# B&R Automation Studio project BR_ZBM1 (part 3)

#### SC_9Init.st - Initialization code
```iecst
(********************************************************************
 * COPYRIGHT --
 ********************************************************************
 * Program: SC_2
 * File: SC_2Init.st
 * Author: ronspa
 * Created: February 16, 2015
 ********************************************************************
 * Implementation of program SC_2
 ********************************************************************)

PROGRAM _INIT

	i := 8;

END_PROGRAM
```

- SC.st (reference to Logical/BunchUnits/SC_Ref/SC.st)

- SC.var (reference to Logical/BunchUnits/SC_Ref/SC.var)

### Program Logical/BunchUnits/BU_10 (IEC) - Program for Bunch Unit 10

#### BU_10Init.st - Initialization code
```iecst
(********************************************************************
 * COPYRIGHT --
 ********************************************************************
 * Program: BU_1
 * File: BU_1Init.st
 * Author: ronspa
 * Created: Januari 12, 2015
 ********************************************************************
 * Implementation of program BU_1
 ********************************************************************)

PROGRAM _INIT

	i := 9;

	BU[i].typInterface.Status := BU_ST_DISABLED;
	BU[i].usChainPos := SHFTREG.uiBunchUnitPosition[i] - 1; // Because position is 0!!!

	// For TESTING RSP 23-12-2014

	//Enable 'FI'
	BU[i].typBunchBelts.command.bEnabledStop := TRUE;
	//Bepaal draairichting
	BU[i].typBunchBelts.command.bRunReverse := FALSE;
	BU[i].typSettings.usTimingBU16 := 14; // Pos=0 ->

END_PROGRAM
```

- BunchUnit.st (reference to Logical/BunchUnits/BU_Ref/BunchUnit.st)

- BunchUnit.var (reference to Logical/BunchUnits/BU_Ref/BunchUnit.var)

### Program Logical/BunchUnits/SC_10 (IEC) - Program for Servo 10

#### SC_10Init.st - Initialization code
```iecst
(********************************************************************
 * COPYRIGHT --
 ********************************************************************
 * Program: SC_2
 * File: SC_2Init.st
 * Author: ronspa
 * Created: February 16, 2015
 ********************************************************************
 * Implementation of program SC_2
 ********************************************************************)

PROGRAM _INIT

	i := 9;

END_PROGRAM
```

- SC.st (reference to Logical/BunchUnits/SC_Ref/SC.st)

- SC.var (reference to Logical/BunchUnits/SC_Ref/SC.var)

### Package Logical/Exceptionhandling - All error codes and exceptions

### Program Logical/Exceptionhandling/ErrorHandling (IEC) - Program

#### ErrorHandling.st - Implementation code
```iecst
(********************************************************************
 * COPYRIGHT --
 ********************************************************************
 * Program: ErrorHandling
 * File: ErrorHandling.st
 * Author: jorkes
 * Created: July 21, 2014
 ********************************************************************
 * Implementation of program ErrorHandling
 ********************************************************************)

PROGRAM _INIT

(* TODO : Add your code here *)

END_PROGRAM

PROGRAM _CYCLIC
	tonHeartBeat( IN:= NOT(EDGE(bHeartBeat)), PT:= INT_TO_TIME(Settings.HeartBeatTime));
	IF EDGE(tonHeartBeat.Q ) THEN
		// LOG
		IF(tonHeartBeat.Q) THEN
			AsArLogWrite_Failed(enable := TRUE, ident := arlogBASE_USER_LOG_IDENT, logLevel := 1, errornr := 50001, mem := 0, len := 0, asciiString :=  ADR('Heart beat failed!!!!'));
		ELSE
			AsArLogWrite_Restored(enable := TRUE, ident := arlogBASE_USER_LOG_IDENT, logLevel := 1, errornr := 50001, mem := 0, len := 0, asciiString :=  ADR('Heart beat active again'));
		END_IF
	END_IF

	IF MCU.typIN.bEmergencyStop THEN
		ErrorState := EMERGENCYSTOP;
	ELSIF MCU.typIN.bDoorOpen THEN
		ErrorState := DOOROPEN;
	ELSIF MCU.typIN.bServiceMode THEN
		ErrorState := SERVICEMODE;
	ELSIF MCU.typIN.bAirpressure THEN
		ErrorState := AIRPRESSURE;
	ELSIF MCU.typIN.bBinder THEN
		ErrorState := BINDER;
	ELSE
		ErrorState := OK;
	END_IF

	//enumError
	CASE ErrorState OF
		0: bGblRun := FALSE;//EmergencyStop
		1: //AirPressure
		2: //DoorOpen
		3: //MotorMalfunction
		4: //Communication
		5: //Binder
		6: //ServiceMode
	END_CASE

END_PROGRAM
```

#### ErrorHandling.var - Local variables
```iecst
(********************************************************************
 * COPYRIGHT --
 ********************************************************************
 * Program: ErrorHandling
 * File: ErrorHandling.var
 * Author: jorkes
 * Created: July 21, 2014
 ********************************************************************
 * Local variables of program ErrorHandling
 ********************************************************************)
VAR
	tonHeartBeat : TON;
	bHeartBeat : BOOL;
	AsArLogWrite_Failed : AsArLogWrite := (0);
	AsArLogWrite_Restored : AsArLogWrite := (0);
	LogMsg : STRING[80];
END_VAR
```

### Program Logical/Exceptionhandling/can_diag (IEC) - Program

#### can_diag.st - Implementation code
```iecst
(********************************************************************
 * COPYRIGHT -- Bernecker + Rainer
 ********************************************************************
 * Program: can_diag
 * File: can_diag.st
 * Author: fleischerm
 * Created: February 02, 2015
 ********************************************************************
 * Implementation of program can_diag
 ********************************************************************)

//******************************************************************
//
//	i n i t
//
//******************************************************************
PROGRAM _INIT

//******************************************************************
// RCX Common Status & Errors Codes
//------------------------------------------------------------------
// variable for the following error codes is -> x20if1041map.comError
//------------------------------------------------------------------
//	RCX_S_OK						0x00000000	Success, Status Okay
//	RCX_E_FAIL						0xC0000001 	Fail
//	RCX_E_UNEXPECTED				0xC0000002	Unexpected
//	RCX_E_OUTOFMEMORY				0xC0000003 	Out OF Memory
//	RCX_E_UNKNOWN_COMMAND			0xC0000004	Unknown Command
//	RCX_E_UNKNOWN_DESTINATION		0xC0000005	Unknown Destination
//	RCX_E_UNKNOWN_DESTINATION_ID	0xC0000006	Unknown Destination ID
//	RCX_E_INVALID_PACKET_LEN		0xC0000007	Invalid Packet Length
//	RCX_E_INVALID_EXTENSION			0xC0000008	Invalid Extension
//	RCX_E_INVALID_PARAMETER			0xC0000009	Invalid Parameter
//	RCX_E_WATCHDOG_TIMEOUT			0xC000000C	Watchdog Timeout
//	RCX_E_INVALID_LIST_TYPE			0xC000000D	Invalid List Type
//	RCX_E_UNKNOWN_HANDLE			0xC000000E	Unknown Handle
//	RCX_E_PACKET_OUT_OF_SEQ			0xC000000F	Out OF Sequence
//	RCX_E_PACKET_OUT_OF_MEMORY		0xC0000010	Out OF Memory
//	RCX_E_QUE_PACKETDONE			0xC0000011	Queue Packet Done
//	RCX_E_QUE_SENDPACKET			0xC0000012	Queue Send Packet
//	RCX_E_POOL_PACKET_GET			0xC0000013	Pool Packet Get
//	RCX_E_POOL_GET_LOAD				0xC0000015	Pool Get Load
//	RCX_E_REQUEST_RUNNING			0xC000001A	Request Already Running
//	RCX_E_INIT_FAULT				0xC0000100	Initialization Fault
//	RCX_E_DATABASE_ACCESS_FAILED	0xC0000101	Database ACCESS Failed
//	RCX_E_NOT_CONFIGURED			0xC0000119	NOT Configured
//	RCX_E_CONFIGURATION_FAULT		0xC0000120	Configuration Fault
//	RCX_E_INCONSISTENT_DATA_SET		0xC0000121	Inconsistent Data Set
//	RCX_E_DATA_SET_MISMATCH			0xC0000122	Data Set Mismatch
//	RCX_E_INSUFFICIENT_LICENSE		0xC0000123	Insufficient License
//	RCX_E_PARAMETER_ERROR			0xC0000124	Parameter Error
//	RCX_E_INVALID_NETWORK_ADDRESS	0xC0000125	Invalid Network Address
//	RCX_E_NO_SECURITY_MEMORY		0xC0000126	No Security Memory
//	RCX_E_NETWORK_FAULT				0xC0000140	Network Fault
//	RCX_E_CONNECTION_CLOSED			0xC0000141	Connection Closed
//	RCX_E_CONNECTION_TIMEOUT		0xC0000142	Connection Timeout
//	RCX_E_LONELY_NETWORK			0xC0000143	Lonely Network
//	RCX_E_DUPLICATE_NODE			0xC0000144	Duplicate Node
//	RCX_E_CABLE_DISCONNECT			0xC0000145	Cable Disconnected
//	RCX_E_BUS_OFF					0xC0000180	Network Node Bus Off
//	RCX_E_CONFIG_LOCKED				0xC0000181	Configuration Locked
//	RCX_E_APPLICATION_NOT_READY		0xC0000182	Application NOT Ready
//	RCX_E_TIMER_APPL_PACKET_SENT	0xC002000C	Timer App Packet Sent
//******************************************************************

//******************************************************************
// RCX Status & Error Codes Slave State
//------------------------------------------------------------------
// variable for the following error codes is -> x20if1041map.slaveState
//------------------------------------------------------------------
//	RCX_SLAVE_STATE_UNDEFINED		0x00000000	UNDEFINED
//	RCX_SLAVE_STATE_OK				0x00000001	OK
//	RCX_SLAVE_STATE_FAILED			0x00000002	FAILED (at least one slave)
//******************************************************************

//******************************************************************
// init some variables
//******************************************************************
step									:= 255;
getDiagInfo								:= FALSE;

END_PROGRAM

//******************************************************************
//
//	c y c l i c
//
//******************************************************************
PROGRAM _CYCLIC

	//******************************************************************************
	// Havatec global used data structure for OPC, VIS and Control
	//**************************************************************
	BU[0];

	//******************************************************************************
	// CANopen Master -> X20IF1041-1
	// get data structure from the I/O mapping
	//**************************************************************
	CASE x20if1041map.comState OF
	//**************************************************************
	0: 	// Unkown
	2:	// Stop
	3:	// Standby
	4:	// Operate
	END_CASE

	//**************************************************************
	CASE x20if1041map.comError OF
	//**************************************************************
	16#C0000140:	// General communication error (this error will occur if at least one slave in the CAN network isn't working)
	16#C0000142:	// Timeout while establishing connection
	16#C0000144:	// Repeated node number found in CAN network
	16#C0000145:	// CAN cable has been disconnected
	END_CASE

	//**************************************************************
	CASE x20if1041map.slaveState OF
	//**************************************************************
	0: 	// Undefined
	1:	// OK
	2:	// Failed
	3:	// Warning
	END_CASE

	//******************************************************************************
	// Servo Unit I/O mapping
	// - Module OK signal
	// - will be FALSE on network or cable error
	//**************************************************************
	IF (BU[0].typServo.bOnLine = FALSE) THEN							// a better check is to wait a certain time before the error is TRUE
		;
	END_IF

	//**************************************************************
	// Servo Unit I/O mapping
	// - Festo drive in error state
 	// -- 16#08 means drive is faulty
	//**************************************************************
	IF (BU[0].typServo.packed.SCON.3 = TRUE) THEN
		getDiagInfo						:= TRUE;
	ELSE
		getDiagInfo						:= FALSE;
	END_IF

	//**************************************************************
	IF EDGEPOS(getDiagInfo) THEN
		step							:= 2;							// next step -
	END_IF

	//******************************************************************************
	// call different function blocks
	//**************************************************************
	CASE step OF														// case function switch of
	//**************************************************************
	1:	// get emergency telegrams
		//**********************************************************
		nxcomRecvEmcyDev_0.enable 		:= TRUE;						// enable function block
		nxcomRecvEmcyDev_0.pDevice 		:= ADR('SS1.IF1');				// CANopen interface address
		nxcomRecvEmcyDev_0.node 		:= 3;							// node number (client address)
		nxcomRecvEmcyDev_0.flags		:= nxcomFLAG_PEEK;				// means: Don't remove node from the diagnostics list
		nxcomRecvEmcyDev_0.pEmcyData	:= ADR(emcyTelegram);			// pointer to an array of 5 emergency telegrams with 8 bytes each
		nxcomRecvEmcyDev_0();											// call function block instance

		//**********************************************************
		CASE nxcomRecvEmcyDev_0.status OF								// case function switch of
		//**********************************************************
		65535:	// ERR_BUSY
			//******************************************************
			;															// wait for different status
		//**********************************************************
		0:		// ERR_OK
			//******************************************************
			nxcomRecvEmcyDev_0.coStatus;								// see help file for the nxcomGetDiag function block
			nxcomRecvEmcyDev_0.emcyCount;								// ...
			//******************************************************
			step						:= 255;							// next step -
		ELSE
			//******************************************************
			step						:= 255;							// next step -
		END_CASE

	//**************************************************************
	2:	// read the diagnostics for the specified node
		// ->
		// -> inclusive the last b5 emergency telegrams
		// ->
		//**********************************************************
		nxcomGetDiag_0.enable 			:= TRUE;						// enable function block
		nxcomGetDiag_0.pDevice 			:= ADR('SS1.IF1');				// CANopen interface address
		nxcomGetDiag_0.node 			:= 3;							// node number (client address)
		nxcomGetDiag_0.flags 			:= nxcomFLAG_PEEK;				// means: Don't remove node from the diagnostics list
		nxcomGetDiag_0.pEmcyData 		:= ADR(emcyTelegram);			// pointer to an array of 5 emergency telegrams with 8 bytes each
		nxcomGetDiag_0();												// call function block instance

		//**********************************************************
		CASE nxcomGetDiag_0.status OF									// case function switch of
		//**********************************************************
		65535:	// ERR_BUSY
			//******************************************************
			;															// wait for different status
		//**********************************************************
		0:		// ERR_OK
			//******************************************************
			nxcomGetDiag_0.coStatus;									// see help file for the nxcomGetDiag function block
			nxcomGetDiag_0.nodeFlags;									// ...
			nxcomGetDiag_0.lastDiagInfo;								// ...
			nxcomGetDiag_0.devType;										// ...
			nxcomGetDiag_0.nmtState;									// ...
			nxcomGetDiag_0.emcyCount;									// Number of actually read emergency telegrams.
			//******************************************************
			step						:= 255;							// next step -
		ELSE
			//******************************************************
			step						:= 255;							// next step -
		END_CASE
	ELSE
		//**********************************************************
		step							:= 255;							// next step -
	END_CASE

END_PROGRAM

//******************************************************************
//
//	e x i t
//
//******************************************************************
PROGRAM _EXIT

//******************************************************************
// TODO : Add your code here
//******************************************************************
nxcomRecvEmcyDev_0.enable 				:= FALSE;						// disable function block on exit
nxcomRecvEmcyDev_0();													// call function block instance

//******************************************************************
nxcomGetDiag_0.enable 					:= FALSE;						// disable function block on exit
nxcomGetDiag_0();														// call function block instance

END_PROGRAM
```

#### can_diag.typ - Local data types
```iecst
(********************************************************************
 * COPYRIGHT -- Bernecker + Rainer
 ********************************************************************
 * Program: can_diag
 * File: can_diag.typ
 * Author: fleischerm
 * Created: February 02, 2015
 ********************************************************************
 * Local data types of program can_diag
 ********************************************************************)

TYPE
	local_if1041_map : 	STRUCT
		comCOS : UDINT;
		comState : UDINT;
		comError : UDINT;
		version : UINT;
		watchdogTimeout : UINT;
		watchdogHost : UDINT;
		errorCount : UDINT;
		errorLogIndicator : UDINT;
		slaveState : UDINT;
		slaveErrorLogIndicator : UDINT;
		slavesConfigured : UDINT;
		slavesActive : UDINT;
		slavesFaulted : UDINT;
	END_STRUCT;
END_TYPE
```

#### can_diag.var - Local variables
```iecst
(********************************************************************
 * COPYRIGHT -- Bernecker + Rainer
 ********************************************************************
 * Program: can_diag
 * File: can_diag.var
 * Author: fleischerm
 * Created: February 02, 2015
 ********************************************************************
 * Local variables of program can_diag
 ********************************************************************)
VAR
	getDiagInfo : BOOL;
	step : USINT;
	x20if1041map : local_if1041_map;
	emcyTelegram : nxcomEmcyTelegrams_t;
	nxcomGetDiag_0 : nxcomGetDiag;
	nxcomRecvEmcyDev_0 : nxcomRecvEmcyDev;
END_VAR
```

- Visualisation Logical/Visualisation (not shown)

### Package Logical/Docs - Package

### ToDo.txt
```
In BunchUnit Ref is de aanstuur tijde van de puls aangepast van 100 -> 1000 voor test.

Bij tijdelijke code van Ronald staat de aanduiding RSPA, dit moet voor de uit eindelijk versie recht gezet worden.

Lijst van openstaande punten:

- Het afvoer bit implementeren zodat de BU geleegd kan worden.
- De timing voor de BunchBelt control in valiabele zetten
- CAN-bus communicatie check
- Keep alive met OPC implementeren, ter indicatie of de PC leeft (Actie bedenken indien dood)
- Enable koppelen aan VNC GUI, zodat met minder BU's gewerkt kan worden.
- GUI aanpassen zodat deze door de lijst van BU's kan lopen.
- Aansturing MBU
- Error handling

Upzoeken.

- Hoe worden de instellingen van een frequency regelaar opgeslagen? o.a adres, ACC, DEC, LSP HSP
```

- brwebSvr.cfg (not shown)

- env.asp (not shown)

### env.asp.txt
(txt body not rendered)

- pv.asp (not shown)

### pv.asp.txt
(txt body not rendered)

- temperature.asp (not shown)

- temperature.svg.asp (not shown)

### temperature.svg.asp.txt
(txt body not rendered)

- webprint.asp (not shown)

### webprint.asp.txt
(txt body not rendered)

- error.txt.asp (not shown)

### login.html.txt
(txt body not rendered)

### logout.html.txt
(txt body not rendered)

- userrights.txt.asp (not shown)

- goform.asp (not shown)

### goform.asp.txt
(txt body not rendered)

- multi.asp (not shown)

- start.asp (not shown)

### start.asp.txt
(txt body not rendered)

### index.html.txt
```
html:
  head:
    title = My Window Title
  body:
    h1 = My Title
    p = My text passage.
```

- ASP_Access.jar (binary file, 10554 bytes)
- BR_ASP_Request.java (not shown)

### coffee_extract.svg.txt
```
svg (font-size=13.3333, font-family=Arial Unicode MS, Sans-serif, preserveAspectRatio=XMidYMid meet, width=100%, height=100%, viewBox=0 0 400 400, text-rendering=geometricPrecision)
  script ({http://www.w3.org/1999/xlink}href=/PV_Access.js, type=text/javascript)
  style = .txGroupTitle{ fill:rgb( 77, 77, 77 ); font-weight:bold  }
			.clBackGradientOwer{ fill:rgb( 26, 26, 26 ); }
			.clOutline{ stroke:rgb(89,89,89); }
			.clHeaderBar{ fill:rgb( 204, 204, 204 ); }
			.clGroupBackground{ fill:rgb( 242, 242, 242 ); }
			.gdBackGradientUpper{ stop-color:rgb( 217, 217, 217 ); }
			.gdBackGradientOwer{ stop-color:rgb( 26, 26, 26 ); }
			.gdControlActiveArea{ stop-color:rgb( 230, 230, 230 ); } (type=text/css)
  script = var list = new Array();
		var actIndex= 0;
		var that = this;
		
		// Example cyclic update request for registered PVs in list. 
		// one PV value requested per call
		refreshPV = function()
		{
			if(list[0] == null) return;  

			actIndex++;        
			if(actIndex >= list.length) 
			{
				actIndex = 0;
			}
			var tmp = list[actIndex];
			 
			pvAccess.ReadPV( tmp[0].getAttribute(tmp[1]), tmp);

		}
		
		// make the changes visible in the document
		refreshPVupdate = function()
		{
			if(list[0] == null) return;  
			
			for(i = 0 ; i <= list.length-1; i++ )
			{
			var temp = list[i];
			temp[0].setAttribute(temp[2], temp[3] );
			temp[0][temp[2]] = temp[3];
			}

		}
		

		
		// registration example
		registerRefreshPV = function(node,nameAttrib,valueAttrib) 
		{
			tmp = new Array();
			tmp.push(node);
			tmp.push(nameAttrib);
			tmp.push(valueAttrib);
			tmp.push(null);
			list.push(tmp);
		}
  defs:
    linearGradient buttonArea (x1=0.5, y1=0, x2=0.5, y2=1)
      stop (offset=0, class=gdBackGradientUpper)
      stop (offset=0.2, class=gdControlActiveArea)
      stop (offset=0.8, class=gdControlActiveArea)
      stop (offset=1, class=gdBackGradientOwer)
  g (transform=translate(100,20), font-size=13.3333)
    rect (x=0, y=0, width=200, height=113, rx=2, ry=2, class=clGroupBackground)
    rect (x=2, y=2, width=198, height=23, class=clHeaderBar)
    text = Control (x=10, y=18, class=txGroupTitle, font-size=12)
    line (x1=0, x2=200, y1=25, y2=25, class=clOutline)
    rect (x=0, y=0, width=200, height=113, rx=2, ry=2, fill=none, class=clOutline)
    g (transform=translate(0,25))
      g (onclick=pvAccess.WritePV('gMainLogic.cmd.switchOnOff','1');, transform=translate(10,10))
        rect (x=1, y=1, width=91, height=31, class=clBackGradientOwer, rx=2, ry=2)
        g:
          rect (x=0.5, y=0.5, width=90, height=30, fill=url(#buttonArea), class=clOutline, rx=2, ry=2)
          text = On (x=45, y=21, text-anchor=middle, class=txGroupTitle)
      g (onclick=pvAccess.WritePV('gMainLogic.cmd.switchOnOff','0');, transform=translate(10,46))
        rect (x=1, y=1, width=91, height=31, class=clBackGradientOwer, rx=2, ry=2)
        g:
          rect (x=0.5, y=0.5, width=90, height=30, fill=url(#buttonArea), class=clOutline, rx=2, ry=2)
          text = Off (x=45, y=21, text-anchor=middle, class=txGroupTitle)
      circle gMainLogic.cmd.switchOnOff (id=machineStatus, cx=160, cy=43, r=10, fill=red)
  text = gBrewing.status.brewingStepText: (x=100, y=180)
  text gBrewing.status.brewingStepText = - (x=100, y=200, id=szTemp)
  text = Each second one update for a PV Value is requested. (x=100, y=240, fill=grey)
  text = Here are two PV's in a cylic update list, so an (x=100, y=260, fill=grey)
  text = update may need two seconds to become visible. (x=100, y=280, fill=grey)
  script = // change color of  status led 
			statusNode = document.getElementById("machineStatus"); 
			function update() { 
				if(statusNode.value ==1) { statusNode.setAttribute("fill", "green"); } 
				else { statusNode.setAttribute("fill", "red"); }; 
			} 	
			

			// register PVs attached to an Element (See line 116 and 124 )
			registerRefreshPV(document.getElementById('machineStatus'), "name","value");
			registerRefreshPV(document.getElementById('szTemp'), "name","textContent");
			
			// periodically called functions (time in ms)
			var refreshInterval  = setInterval("refreshPV();" ,1000);
			var refreshInterval2 = setInterval("refreshPVupdate();", 100);			
			var updateInterval   = setInterval("update();",10);
```

### JS_Demo.htm.txt
(txt body not rendered)

- response.asp (not shown)

- ASP-Access.exe (binary file, 10752 bytes)
### br_ASPGoform.cs
```
using System;
using System.Collections.Generic;
using System.Linq;
using System.Text;
using System.Net;
using System.IO;

namespace BR_ASP_Request
{
    public class PV_Access
    {
        private static String pvAccess(String host, String payload)
        {
            string url = "http://" + host + "/goform/ReadWrite";
            byte[] parameter = Encoding.UTF8.GetBytes(payload);
            HttpWebRequest request = (HttpWebRequest)WebRequest.Create(url);
            request.Method = "POST";
            request.Timeout = 3000; // 3 Sek Timeout
            try
            {
                Stream requestStream = request.GetRequestStream();
                requestStream.Write(parameter, 0, parameter.Length);
                requestStream.Close();
                HttpWebResponse response = (HttpWebResponse)request.GetResponse();
                if (response == null) return "";
                Stream responseStream = response.GetResponseStream();
                StreamReader streamReader = new StreamReader(responseStream);
                string antwort = streamReader.ReadToEnd();
                streamReader.Close();
                responseStream.Close();
                antwort = antwort.Replace("<!-- B&R ASP Webserver -->", "");
                return antwort;
            }
            catch (Exception e)
            {
                return e.Message;
            }
        }

        public static String ReadPV(String host, String PvName)
        {
            string Parameter = "redirect=/response.asp&read=1&variable=" + PvName + "&value=none";
            return pvAccess(host, Parameter);
        }

        public static String WritePV(String host, String PvName, String PvValue)
        {
            string Parameter = "redirect=/response.asp&write=1&variable=" + PvName + "&value=" + PvValue;
            return pvAccess(host, Parameter);
        }
    }
}
```

### Package Logical/IOHandling - Package

### Program Logical/IOHandling/IOpolling (IEC) - Program

#### IOpolling.st - Implementation code
```iecst
(********************************************************************
 * COPYRIGHT -- Microsoft
 ********************************************************************
 * Program: IOpolling
 * File: IOpolling.st
 * Author: jorkes
 * Created: October 24, 2014
 ********************************************************************
 * Implementation of program IOpolling
 ********************************************************************)

PROGRAM _INIT

END_PROGRAM

PROGRAM _CYCLIC

	ElevatorCil(BU[0], BU[i].typIN.bElevatorUp, BU[i].typIN.bElevatorMid, BU[i].typIN.bElevatorDown);

END_PROGRAM
```

#### IOpolling.var
```iecst
VAR
	i : USINT;
	Down_SR : SR;
	Mid_SR : SR;
	Up_SR : SR;
	bDown : BOOL;
	bMid : BOOL;
	bUp : BOOL;
	EnumInput : enum_Input;
END_VAR
```

#### IOpolling.typ - Local data types
```iecst
(********************************************************************
 * COPYRIGHT -- Microsoft
 ********************************************************************
 * Program: IOpolling
 * File: IOpolling.typ
 * Author: jorkes
 * Created: October 27, 2014
 ********************************************************************
 * Local data types of program IOpolling
 ********************************************************************)

TYPE
	enum_Input :
		(
		CILUP := 3,
		CILMID := 4,
		CILDOWN := 5
		);
END_TYPE
```

### Package Logical/Lichtkrant - Read and write serial Frames

### Program Logical/Lichtkrant/Sender (IEC) - sending serial data

#### SenderCyclic.st - Cyclic code
```iecst
(********************************************************************
 * COPYRIGHT -- Bernecker + Rainer
 ********************************************************************
 * Program: Sender
 * File: SenderCyclic.st
 * Author: Bernecker & Rainer
 * Created: January 25, 2010
 ********************************************************************
 * Implementation of program Sender
 ********************************************************************)

(*************init program**********************)
PROGRAM _INIT
	serial_0.enable := TRUE;												(*enable sender by default*)
END_PROGRAM

(*************cyclic program********************)
PROGRAM _CYCLIC

	txtChainCounter := UINT_TO_STRING(SHFTREG.typCounters.usChainCounter);
	txtSubChainCounter := UINT_TO_STRING(SHFTREG.typCounters.usChainOffset);

	text1 := CONCAT('cnt: ', txtChainCounter);
	text1 := CONCAT(text1, ' ');
	text1 := CONCAT(text1, 'sub: ');
	text1 := CONCAT(text1, txtSubChainCounter);
	IF RU.typOUT.bActivateGripper THEN
		text1 := 'Reject active!!!';
	END_IF

	IF BU[0].typOUT.bActivateGripper THEN
		text1 := 'BU -0-';
	END_IF
	IF BU[1].typOUT.bActivateGripper THEN
		text1 := 'BU -1-';
	END_IF
	IF BU[2].typOUT.bActivateGripper THEN
		text1 := 'BU -2-';
	END_IF
	IF BU[3].typOUT.bActivateGripper THEN
		text1 := 'BU -3-';
	END_IF
	IF BU[4].typOUT.bActivateGripper THEN
		text1 := 'BU -4-';
	END_IF
	IF BU[5].typOUT.bActivateGripper THEN
		text1 := 'BU -5-';
	END_IF
	IF BU[6].typOUT.bActivateGripper THEN
		text1 := 'BU -6-';
	END_IF
	IF BU[7].typOUT.bActivateGripper THEN
		text1 := 'BU -7-';
	END_IF
	IF BU[8].typOUT.bActivateGripper THEN
		text1 := 'BU -8-';
	END_IF
	IF BU[9].typOUT.bActivateGripper THEN
		text1 := 'BU -9-';
	END_IF

	setText_0.ThisData := LichtkrantData;

	IF Var2 = 1 THEN
		setText_0(font := LichtkrantData.fontCode_.narowSize_4x7);
	ELSIF Var2 = 2 THEN
		setText_0(font := LichtkrantData.fontCode_.normalSize_5x7);
	ELSIF Var2 = 3 THEN
		setText_0(color := LichtkrantData.colorCode_.brightGreen);
	ELSIF Var2 = 4 THEN
		setText_0(color := LichtkrantData.colorCode_.brightOrange);
	ELSIF Var2 = 5 THEN
		setText_0(presentation := LichtkrantData.laggingCom_.upDown);
	ELSIF Var2 = 6 THEN
		setText_0(presentation := LichtkrantData.laggingCom_.horizontalScroll);
	ELSIF Var2 = 7 THEN
		setText_0(presentation := LichtkrantData.laggingCom_.normal);
	ELSIF Var2 = 8 THEN
		setText_0(interval := LichtkrantData.methodSpeed_.fast);
	ELSIF Var2 = 9 THEN
		setText_0(interval := LichtkrantData.methodSpeed_.middle);
	ELSIF Var2 = 10 THEN
		setText_0(interval := LichtkrantData.methodSpeed_.slow);
	END_IF
	Var2 := 0;

	IF text_old <> text1 THEN
		setText_0(IN := text1); //Data conversion
		serial_0(text := setText_0.OUT);
		text_old := text1;
	END_IF

END_PROGRAM
```

#### Sender.var - Local variables
```iecst
(********************************************************************
 * COPYRIGHT -- Bernecker + Rainer
 ********************************************************************
 * Program: Sender
 * File: Sender.var
 * Author: Bernecker & Rainer
 * Created: January 25, 2010
 ********************************************************************
 * Local variables of program Sender
 ********************************************************************)
VAR
	Var2 : USINT := 0;
	serial_0 : fbSerial;
	setText_0 : fbSetText;
	LichtkrantData : DataPackage;
	text_old : STRING[80];
	text1 : STRING[80];
	txtSubChainCounter : STRING[80];
	txtChainCounter : STRING[80];
END_VAR
```

### Package Logical/libraries_hav - Havatec libraries

### Library Logical/libraries_hav/Inverter (IEC, version 3.00.0) - Freq. Inverter Library

#### ACPinverter.st
```iecst
(********************************************************************
 * COPYRIGHT -- Microsoft
 ********************************************************************
 * Library: Inverter
 * Author: HD
 * Created: March 15, 2011
 ********************************************************************
 * Implementation of library Invertor
 ********************************************************************)
(*-------------------------------------------------------------
Setting in I/O configuration X64 ACOPOS inverter

SDC settings	no
IO mapping 	packed

ACPinverter.packed.ETAD		status
ACPinverter.packed.CMDD		command
ACPinverter.packed.LFR		speed [hz]

---------------------------------------------------------------
Com_typ		input		structure
---------------------------------------------------------------
command.iSetSpeed;				[INT]	Hz (0.1) / Rpm (1000 uints = 6 hz) , (+value = forward,  -value = reverse)
command.bPower;					[BOOL]	Power on
command.bEnabledStop			[BOOL]	0 = inverter switch to status "switch on" (16#0023) after stop
																	1 = inverter remain on status "enable operation" (16#0027) after stop
command.bRun;					[BOOL]	Start run forward with value iSetSpeed;
command.bRunReverse;			[BOOL]	Start run reverse with value iSetSpeed;
command.bQuickStop;				[BOOL]	Quickstop, emergency stop
command.bResetFault;			[BOOL]	Reset error on invertor

---------------------------------------------------------------
Sts_typ		output		structure
---------------------------------------------------------------
status.uiDrive;					[UINT]	Drive status (ETAD AND mask 16#006F)
status.bReadyToSwitchOn			[BOOL]	Drive is ready to switch power on
status.bDriveReady;				[BOOL]	Drive is switched on, power is on
status.bRun;					[BOOL]	Drive is running
status.bSetSpeedReached			[BOOL]	Speed setpoint is reached
status.bFault;					[BOOL]	Error active
status.bQuickStopActive;		[BOOL]	Quickstop active
strHmiInfo						[STRING[80]		Hmi info text
strErrorInfo					[STRING(80)]	Fault info text

---------------------------------------------------------------
History:
Version:	Date:				author:	change:
1.00		19-07-2011		HD			changed to one motor structure VAR INOUT
2.00		23-12-2011		HD			added "MotorStruc.status.bSetSpeedReached"
2.10		23-07-2012		HD			when operation enabled, stop then goto switch on
2.20		12-09-2012		HD			Oneshot bit added at reset fault
3.00		07-05-2013		HD			changed and tested for all invertors
3.10		26-06-2013		HD			add fault info "strErrorInfo"	and HMI info "strHmiInfo"
--------------------------------------------------------------- *)

FUNCTION_BLOCK ACPinverter

	IF EDGEPOS(bResetFault) THEN
		_InverterCommand := INV_CMD_INIT;
		bResetFault := FALSE;
	END_IF

	IF iSpeed <> 0 AND iSpeed <> MotorStruc.command.iSetSpeed THEN
		MotorStruc.command.iSetSpeed := iSpeed;
	END_IF

	CASE _InverterCommand OF
		//======================================
		INV_CMD_INIT:
			//======================================
			_InverterCommand := INV_CMD_SETSPEED;
			tonTimeOut.PT := T#500ms;

		//======================================
		INV_CMD_SETSPEED:
			//======================================
			//Set speed (iSetSpeed/30=Hz)
			MotorStruc.command.iSetSpeed := (iSpeed);
			_InverterCommand := INV_CMD_POWERON;

		//======================================
		INV_CMD_POWERON:
			//======================================
			//Power up frequency inverter
			//Check if 'fi' is Ready for switching on
			tonTimeOut(IN := TRUE);

			IF MotorStruc.status.bReadyToSwitchOn THEN
				//Power up 'fi'
				MotorStruc.command.bPower := TRUE;
				_InverterCommand := INV_CMD_READY;
				tonTimeOut(IN := FALSE);
			ELSIF MotorStruc.status.bDriveReady THEN
				_InverterCommand := INV_CMD_READY;
			ELSIF tonTimeOut.Q THEN
				//Power down 'fi'
				MotorStruc.command.bPower := FALSE;
				_InverterCommand := INV_CMD_RESETFAULT;
				tonTimeOut(IN := FALSE);
			END_IF

		//======================================
		INV_CMD_RESETFAULT:
			//======================================
			tonTimeOut(IN := TRUE);
			//Reset fault
			MotorStruc.command.bResetFault := MotorStruc.status.bFault;

			_InverterCommand := INV_CMD_READY;
			//Check for any FAULTS
			IF MotorStruc.status.bFault AND tonTimeOut.Q THEN
				//Stop 'fi'
				MotorStruc.command.bRun := FALSE;
				MotorStruc.status.bRun := FALSE;
				//bRun_ := _bRun;
				MotorStruc.command.bResetFault := FALSE;
				_InverterCommand := INV_CMD_ERROR;
				tonTimeOut(IN := FALSE);
			ELSIF MotorStruc.status.bFault THEN
				MotorStruc.command.bResetFault := TRUE;
			ELSIF tonTimeOut.Q THEN
				tonTimeOut(IN := FALSE);
				_InverterCommand := INV_CMD_INIT;
			END_IF

		//======================================
		INV_CMD_READY:
			//======================================
			tonTimeOut(IN := TRUE);
			InverterState_ := INV_ST_READY;
			//Drive remains in enabled state, when run TRUE or FALSE
			MotorStruc.command.bEnabledStop := TRUE;
			//Check if frequency drive is Ready
			IF MotorStruc.status.bDriveReady THEN
				//'fi' can be operated; bRun, bRunReverse
				MotorStruc.command.bRun := bRun;
				MotorStruc.command.bRunReverse := bRunReverse;
			ELSIF tonTimeOut.Q THEN
				_InverterCommand := INV_CMD_ERROR;
				tonTimeOut(IN := FALSE);
			END_IF

		//======================================
		INV_CMD_ERROR:
			//======================================
			InverterState_ := INV_ST_FAULT;
	END_CASE

	// Speed
	MotorStruc.packed.LFR := MotorStruc.packed.LFRD := MotorStruc.command.iSetSpeed;

	//-------------------------------------------------------------------------------
	// Mask the DRIVECOM status word
	// bit 0 = Ready to switch on
	// bit 1 = Switch on
	// bit 2 = Operation enabled
	// bit 3 = Malfuntion, fault
	// bit 4 = x
	// bit 5 = Quick stop
	// bit 6 = Switch on disabled

	MotorStruc.status.uiDrive := MotorStruc.packed.ETAD AND 16#006F;

	//-------------------------------------------------------------------------------
	MotorStruc.status.bReadyToSwitchOn := 0;
	MotorStruc.status.bDriveReady := 0;
	MotorStruc.status.bRun := 0;
	MotorStruc.status.bQuickStopActive := 0;
	MotorStruc.status.bFault := 0;

	CASE MotorStruc.status.uiDrive OF

		//-------------------------------------------
		16#0000:	// Not ready to switch on
		//-------------------------------------------
		// Error network

		//-------------------------------------------
		16#0007: // Quick stop active
		//-------------------------------------------
		MotorStruc.status.bQuickStopActive := 1;

		// Wait untill quick stop is zero
		IF (MotorStruc.command.bQuickStop = 0) THEN
			MotorStruc.packed.CMDD := 16#0000;
		END_IF

		//-------------------------------------------
		16#0008, 16#0028: // Drive in fault state
		//-------------------------------------------
		MotorStruc.status.bFault := 1;

		// reset fault
		IF (MotorStruc.command.bResetFault = 1) AND (bResetFault = 0) THEN
			MotorStruc.packed.CMDD := 16#0080;
		END_IF
		bResetFault := MotorStruc.command.bResetFault;

		//-------------------------------------------
		16#0040, 16#0050:	// Switch on disable
		//-------------------------------------------
		MotorStruc.status.bReadyToSwitchOn := 1;

		IF (MotorStruc.command.bPower = 1)  THEN
			IF (MotorStruc.command.bQuickStop = 0) THEN
				MotorStruc.packed.CMDD := 16#0006;
			ELSE
				MotorStruc.packed.CMDD := 16#0002;
			END_IF
		ELSE // Disable power
			MotorStruc.packed.CMDD := 16#0000;
		END_IF

		//-------------------------------------------
		16#0021, 16#0031:	// Ready to switch on
		//-------------------------------------------
		IF (MotorStruc.command.bPower = 1)  THEN
			IF (MotorStruc.command.bQuickStop = 0) THEN
				MotorStruc.packed.CMDD := 16#0007;
			ELSE
				MotorStruc.packed.CMDD := 16#0002;
			END_IF
		ELSE // Disable power
			MotorStruc.packed.CMDD := 16#0000;
		END_IF

		//-------------------------------------------
		16#0023:	 // Switch on
		//-------------------------------------------
		MotorStruc.status.bDriveReady := 1;

		//  command run
		IF (MotorStruc.command.bRun = 1) THEN
			IF (MotorStruc.command.bRunReverse = 0) THEN
				MotorStruc.packed.CMDD := 16#000F;
			ELSE//  command run reverse
				MotorStruc.packed.CMDD := 16#080F;
			END_IF
		END_IF

		// Disable power or quick stop
		IF (MotorStruc.command.bPower = 0) THEN
			MotorStruc.packed.CMDD := 16#0000;
		ELSIF (MotorStruc.command.bQuickStop = 1) THEN
			MotorStruc.packed.CMDD := 16#0002;
		END_IF

		//-------------------------------------------
		16#0027: // Operation enabled
		//-------------------------------------------
		MotorStruc.status.bDriveReady := 1;

		//  command run
		IF (MotorStruc.command.bRun = 1) THEN
			MotorStruc.status.bRun := 1;
			IF (MotorStruc.command.bRunReverse = 0) THEN
				MotorStruc.packed.CMDD := 16#000F;
			ELSE//  command run reverse
				MotorStruc.packed.CMDD := 16#080F;
			END_IF
		ELSE // stop
			MotorStruc.status.bRun := 0;
			IF	(MotorStruc.command.bEnabledStop = 1) THEN	// Invertor remains in enable operation status 16#0027
				MotorStruc.packed.CMDD := 16#110F;						// S44 / P74 / P84 = 16#010F, X64 = 16#100F
			ELSE
				MotorStruc.packed.CMDD := 16#0007;	 					// Invertor in switched on status 16#0023
			END_IF
		END_IF

		// Disable power or quick stop
		IF (MotorStruc.command.bPower = 0) THEN
			MotorStruc.packed.CMDD := 16#0000;
		ELSIF (MotorStruc.command.bQuickStop = 1) THEN
			MotorStruc.packed.CMDD := 16#0002;
		END_IF

		ELSE	// status unknown
		MotorStruc.packed.CMDD := 16#0000;

	END_CASE

	MotorStruc.status.bSetSpeedReached := MotorStruc.packed.ETAD.10 AND MotorStruc.status.bRun;

	//--------------------------------------------------------------------------------------------
	// HMI info, drive state
	//--------------------------------------------------------------------------------------------
	CASE MotorStruc.packed.HMIS OF

		1: MotorStruc.status.strHmiInfo := 'DC injection braking (dCb)';
		2: MotorStruc.status.strHmiInfo := 'Drive ready (rdY)';
		3: MotorStruc.status.strHmiInfo := 'Freewheel stop control (nSt)';
		4: MotorStruc.status.strHmiInfo := 'Drive running (rUn)';
		5: MotorStruc.status.strHmiInfo := 'In accel. (ACC)';
		6: MotorStruc.status.strHmiInfo := 'In decel. (dEC)';
		7: MotorStruc.status.strHmiInfo := 'Current limitation (CLI)';
		8: MotorStruc.status.strHmiInfo := 'Fast stop (FSt)';
		9: MotorStruc.status.strHmiInfo := 'Vector regulation active (FLU)';
		11: MotorStruc.status.strHmiInfo := 'Control switched on, DC bus not charged (nLP)';
		12: MotorStruc.status.strHmiInfo := 'Active PWR (PrA)';
		13: MotorStruc.status.strHmiInfo := 'Controlled stop (CtL)';
		14: MotorStruc.status.strHmiInfo := 'Adapted deceleration (Obr)';
		15: MotorStruc.status.strHmiInfo := 'Standby output cut (SOC)';
		17: MotorStruc.status.strHmiInfo := 'Undervoltage alarm (USA)';
		18: MotorStruc.status.strHmiInfo := 'TC indust. mode activated (tC)';
		19: MotorStruc.status.strHmiInfo := 'in autotest (St)';
		20: MotorStruc.status.strHmiInfo := 'autotest error (FA)';
		21: MotorStruc.status.strHmiInfo := 'Autotest OK (YES)';
		22: MotorStruc.status.strHmiInfo := 'eeprom test (EP)';
		23: MotorStruc.status.strHmiInfo := 'In fault (FLt)';
		28: MotorStruc.status.strHmiInfo := 'Safety level SS1 active (SS1)';
		29: MotorStruc.status.strHmiInfo := 'Safety level SLS active (SLS)';
		30: MotorStruc.status.strHmiInfo := 'Safety level STO active (StO)';
	END_CASE

	//--------------------------------------------------------------------------------------------
	// Error info
	//--------------------------------------------------------------------------------------------
	IF (MotorStruc.status.bFault) THEN

		MotorStruc.status.strErrorInfo :='Fault';
		CASE MotorStruc.packed.ERRD OF
			1:	MotorStruc.status.strErrorInfo := 'Calibration error (InF)';
			2:	MotorStruc.status.strErrorInfo := 'Control Eeprom (EEF1)';
			3:	MotorStruc.status.strErrorInfo := 'Internal- I measure (InF9)';
			4:	MotorStruc.status.strErrorInfo := 'Internal-mains circuit (InFA)';
			5:	MotorStruc.status.strErrorInfo := 'Modbus com. (SLF1)';
			6:	MotorStruc.status.strErrorInfo := 'int. com.link (ILF)';
			7:	MotorStruc.status.strErrorInfo := 'Com. network (CnF)';
			8:	MotorStruc.status.strErrorInfo := 'External fault at LI or local connection (EPF1)';
			9:	MotorStruc.status.strErrorInfo := 'Overcurrent (OCF)';
			10:	MotorStruc.status.strErrorInfo := 'Capacitor precharge (CrF)';
			11:	MotorStruc.status.strErrorInfo := 'Encoder feedback signal missing (SPF)';
			16:	MotorStruc.status.strErrorInfo := 'Drive overheat (OHF)';
			17:	MotorStruc.status.strErrorInfo := 'Motor overload (OLF)';
			18:	MotorStruc.status.strErrorInfo := 'Overbraking (ObF)';
			19:	MotorStruc.status.strErrorInfo := 'Mains overvoltage (OSF)';
			20:	MotorStruc.status.strErrorInfo := '1 output phase loss (OPF1)';
			21:	MotorStruc.status.strErrorInfo := 'Input phase loss (PHF)';
			22:	MotorStruc.status.strErrorInfo := 'Mains Undervoltage (USF)';
			23:	MotorStruc.status.strErrorInfo := 'Motor short circuit phase/phase (SCF1)';
			24:	MotorStruc.status.strErrorInfo := 'Motor overspeed (SOF)';
			25:	MotorStruc.status.strErrorInfo := '[Auto-tuning] (tnF)';
			26:	MotorStruc.status.strErrorInfo := 'Unknown drive rating (InF1)';
			27:	MotorStruc.status.strErrorInfo := 'Unknown or incompatible power board (InF2)';
			28:	MotorStruc.status.strErrorInfo := 'Interruption of internal serial communication (InF3)';
			29:	MotorStruc.status.strErrorInfo := 'Invalid industrialization zone (InF4)';
			30:	MotorStruc.status.strErrorInfo := 'Power Eeprom (EEF2)';
			31:	MotorStruc.status.strErrorInfo := 'Impedant sh. circuit (SCF2)';
			32:	MotorStruc.status.strErrorInfo := 'Ground short circuit (SCF3)';
			33:	MotorStruc.status.strErrorInfo := '3 output phase loss (OPF2)';
			34:	MotorStruc.status.strErrorInfo := 'CAN com. (COF)';
			35:	MotorStruc.status.strErrorInfo := 'Brake control (bLF)';
			38:	MotorStruc.status.strErrorInfo := 'External fault com. (EPF2)';
			41:	MotorStruc.status.strErrorInfo := 'Brake feedback (brF)';
			42:	MotorStruc.status.strErrorInfo := 'PC com. (SLF2)';
			43:	MotorStruc.status.strErrorInfo := 'Enc. coupl. (ECF)';
			44:	MotorStruc.status.strErrorInfo := 'Torque/current limit (SSF)';
			45:	MotorStruc.status.strErrorInfo := 'HMI com. (SLF3)';
			46:	MotorStruc.status.strErrorInfo := 'Power removal (PrF)';
			49:	MotorStruc.status.strErrorInfo := 'LI6=PTC probe (PtFL)';
			50:	MotorStruc.status.strErrorInfo := 'PTC fault (OtFL)';
			51:	MotorStruc.status.strErrorInfo := 'Internal- I measure (InF9)';
			52:	MotorStruc.status.strErrorInfo := 'Internal-mains circuit (InFA)';
			53:	MotorStruc.status.strErrorInfo := 'Internal- thermperature sensor (InFb)';
			54:	MotorStruc.status.strErrorInfo := 'IGBT overheat (tJF)';
			55:	MotorStruc.status.strErrorInfo := 'IGBT short circuit (SCF4)';
			56:	MotorStruc.status.strErrorInfo := 'Motor short circuit (SCF5)';
			57:	MotorStruc.status.strErrorInfo := 'Torque time-out (SrF)';
			58:	MotorStruc.status.strErrorInfo := 'Output contactor stuck (closed) (FCF1)';
			59:	MotorStruc.status.strErrorInfo := 'Outut contactor open (FCF2)';
			61:	MotorStruc.status.strErrorInfo := 'AI2 input (AI2F)';
			64:	MotorStruc.status.strErrorInfo := 'input contactor fault (LCF)';
			66:	MotorStruc.status.strErrorInfo := 'Diff. I fault (dCF)';
			67:	MotorStruc.status.strErrorInfo := 'IGBT desaturation (HdF)';
			68:	MotorStruc.status.strErrorInfo := 'Unknown or incompatible option card (InF6)';
			69:	MotorStruc.status.strErrorInfo := 'internal CPU error (InFE)';
			71:	MotorStruc.status.strErrorInfo := 'AI3 4-20mA loss (LFF3)';
			73:	MotorStruc.status.strErrorInfo := 'Error in hardware configuration (HCF)';
			76:	MotorStruc.status.strErrorInfo := 'Dynamic load fault (dLF)';
			77:	MotorStruc.status.strErrorInfo := 'Internal- thermperature sensor (InFb)';
			99:	MotorStruc.status.strErrorInfo := 'Channel switch fault (CSF)';
			100:	MotorStruc.status.strErrorInfo := 'Speed underload (ULF)';
			101:	MotorStruc.status.strErrorInfo := 'Torque Overload Fault (OLC)';
			105:	MotorStruc.status.strErrorInfo := 'Angle error (ASF)';
			107:	MotorStruc.status.strErrorInfo := 'Safety fault (SAFF)';
			108:	MotorStruc.status.strErrorInfo := 'Function Block Errors (FbE)';
			109:	MotorStruc.status.strErrorInfo := 'Function block stop fault (FbES)';

		END_CASE;

	ELSE
		IF NOT MotorStruc.packed.ModuleOk THEN
			MotorStruc.status.strErrorInfo := 'Module error';
		ELSE
			IF MotorStruc.status.bRun THEN
				MotorStruc.status.strErrorInfo := 'Run';
			ELSE
				IF MotorStruc.status.bDriveReady THEN
					MotorStruc.status.strErrorInfo := 'Ready';
				ELSE
					MotorStruc.status.strErrorInfo := '';
				END_IF
			END_IF
		END_IF
	END_IF

END_FUNCTION_BLOCK
```

#### Inverter.typ - Exported data types
```iecst
(********************************************************************
 * COPYRIGHT -- Microsoft
 ********************************************************************
 * Library: Invertor
 * File: Invertor.typ
 * Author: daaneh
 * Created: March 15, 2011
 ********************************************************************
 * Data types of library Invertor
 ********************************************************************)

TYPE
	enumINV_ST :
		(
		INV_ST_READY := 0,
		INV_ST_FAULT := 1,
		INV_ST_RUN := 2
		);
	enumINV_CMD :
		(
		INV_CMD_INIT := 0,
		INV_CMD_SETSPEED := 1,
		INV_CMD_POWERON := 2,
		INV_CMD_RESETFAULT := 3,
		INV_CMD_READY := 4,
		INV_CMD_ERROR := 5
		);
	AcpInverter_typ : 	STRUCT
		command : AcpInverter_command_typ;
		status : AcpInverter_status_typ;
		packed : AcpInverter_packed_typ;
		SDO : SDO_type;
	END_STRUCT;
	AcpInverter_command_typ : 	STRUCT
		iSetSpeed : INT; (*Speed Hz*)
		bPower : BOOL; (*switch drive on*)
		bRun : BOOL; (*run velocity*)
		bRunReverse : BOOL; (*run reverse *)
		bEnabledStop : BOOL;
		bQuickStop : BOOL; (*emergency stop*)
		bResetFault : BOOL; (*reset fault*)
	END_STRUCT;
	AcpInverter_status_typ : 	STRUCT
		uiDrive : UINT; (*drive status 8 bits*)
		bReadyToSwitchOn : BOOL; (*ready for power on*)
		bDriveReady : BOOL; (*power switched on*)
		bRun : BOOL; (*run forward*)
		bSetSpeedReached : BOOL; (*Set speed reached*)
		bQuickStopActive : BOOL; (*emergency stop*)
		bFault : BOOL; (*drive in fault state*)
		strHmiInfo : STRING[80]; (*drive info*)
		strErrorInfo : STRING[80]; (*fault info*)
	END_STRUCT;
	AcpInverter_packed_typ : 	STRUCT
		ETAD : UINT; (*status word*)
		ETI : UINT; (*extended status word*)
		LCR : UINT; (*current 0.1 A*)
		CMDD : UINT; (*command word*)
		CMI : UINT; (*extended command word*)
		ERRD : UINT; (*fault code*)
		HMIS : UINT; (*drive state*)
		RFR : INT; (*output frequentie*)
		RFRD : INT; (*output rpm*)
		OTR : INT; (*Torque %*)
		LFR : INT; (*frequentie setpoint *)
		LFRD : INT; (*Rpm setpoint*)
		LFT : INT; (*last detected fault*)
		ModuleOk : BOOL; (*module OK*)
		Relay : BOOL; (*relay*)
		DigOutput : BOOL; (*digital output*)
	END_STRUCT;
END_TYPE
```

#### Inverter.fun - Exported functions and function blocks
```iecst
(********************************************************************
 * COPYRIGHT -- Microsoft
 ********************************************************************
 * Library: Invertor
 * File: Invertor.fun
 * Author: daaneh
 * Created: March 15, 2011
 ********************************************************************
 * Functions and function blocks of library Invertor
 ********************************************************************)

FUNCTION_BLOCK ACPinverter (*TODO: Add your comment here*)
	VAR_INPUT
		bRun : BOOL;
		bRunReverse : BOOL;
		bResetFault : BOOL;
		iSpeed : INT;
	END_VAR
	VAR_OUTPUT
		InverterState_ : enumINV_ST;
	END_VAR
	VAR_IN_OUT
		MotorStruc : AcpInverter_typ;
	END_VAR
	VAR
		tonTimeOut : TON;
		_InverterCommand : enumINV_CMD;
		zzEdge00000 : BOOL;
	END_VAR
END_FUNCTION_BLOCK
```

### Library Logical/libraries_hav/BULib (IEC) - Bunch Unit library

#### BULib.fun - Exported functions and function blocks
```iecst
(********************************************************************
 * COPYRIGHT --
 ********************************************************************
 * Library: BULib
 * File: BULib.fun
 * Author: ronspa
 * Created: September 29, 2014
 ********************************************************************
 * Functions and function blocks of library BULib
 ********************************************************************)

FUNCTION ElevatorCil : BOOL
	VAR_INPUT
		ThisBU : BunchUnit;
		bUp : BOOL;
		bMid : BOOL;
		bDown : BOOL;
	END_VAR
	VAR
		bElevatorUp_SR : SR;
		bElevatorMid_SR : SR;
		bElevatorDown_SR : SR;
	END_VAR
END_FUNCTION

FUNCTION DefaultSettingsBU : BOOL
	VAR_INPUT
		ThisBU : BunchUnit;
		iHS : USINT;
		iMPD2UL : INT;
		iRP : INT;
		iRlP : INT;
		iSPD : USINT;
		iFSPD : USINT;
		tiDD : TIME;
		tiDRD : TIME;
		uiNCD : UINT;
		iSEPStart : INT := 92;
		iSEPStartVak : INT := 246;
		iSEPEndVak : INT := 443;
		iSEPEnd : INT := 530;
		tiBBP : TIME;
	END_VAR
END_FUNCTION

FUNCTION Elevator : BOOL (*Operate Lift*) (*$GROUP=User*)
	VAR_INPUT
		ThisBU : BunchUnit;
		bElevator : DINT;
	END_VAR
END_FUNCTION

FUNCTION CheckTimers : BU_Status_enum
	VAR_INPUT
		ThisBU : BunchUnit;
		Status : BU_Status_enum;
	END_VAR
	VAR
		tonElevator : TON;
	END_VAR
END_FUNCTION
```

#### BU.typ - Exported data types
```iecst
(********************************************************************
 * COPYRIGHT --
 ********************************************************************
 * File: BU.typ
 * Author: ronspa
 * Created: September 22, 2014
 ********************************************************************
 * Global data types of project The_Magnifica_v0127
 ********************************************************************)

TYPE
	BU_Elevator_enum :
		(
		BU_ELEVATOR_UP := 0,
		BU_ELEVATOR_DOWN := 1
		);
	BU_Visu_Release_enum :
		(
		BU_VISU_RELEASE_OUT := 0,
		BU_VISU_RELEASE_IN := 1
		);
	BU_Visu_Gripper_enum :
		(
		BU_VISU_GRIPPER_OUT := 0,
		BU_VISU_GRIPPER_IN := 1
		);
	BU_Visu_Elevator_enum :
		(
		BU_VISU_ELEVATOR_UP := 0,
		BU_VISU_ELEVATOR_MID := 1,
		BU_VISU_ELEVATOR_DOWN := 2
		);
	BU_Status_enum :
		(
		BU_ST_DISABLED := 0,
		BU_ST_INIT := 1,
		BU_ST_HOME := 2,
		BU_ST_RECEIVE := 3,
		BU_ST_FULL := 4,
		BU_ST_DROPPED := 5,
		BU_ST_RETURN := 6,
		BU_ST_FAILURE := 7,
		BU_ST_TIMEOUT_LIFT := 8,
		BU_ST_TIMEOUT_POSITION := 9,
		BU_ST_MANUAL := 10,
		BU_ST_DROP_POS := 11,
		BU_ST_RECEIVE_POS := 12,
		BU_ST_MOVE_ELEVATOR_UP := 13,
		BU_ST_MOVE_ELEVATOR_DOWN := 14,
		BU_ST_RELEASING := 15,
		BU_ST_WAIT_MCU := 16
		);
	BU_Command_Enum :
		(
		BU_CMD_Ready := 1,
		BU_CMD_Init := 2,
		BU_CMD_Home := 3,
		BU_CMD_Receive := 4,
		BU_CMD_Drop := 5,
		BU_CMD_DropReady := 6,
		BU_CMD_Manual := 7,
		BU_CMD_Hold := 8
		);
	SettingsBU : 	STRUCT
		uiNextChainDelay : UINT := 0; (*Delay in [ms] to enable trigger afther usNextChainInput*)
		iReceivePos : INT := 50;
		iReleasePos : INT := 450;
		usHomeSpeed : USINT := 10; (*Homing speed*)
		usSpeed : USINT := 50; (*Normal servo speed*)
		usFastSpeed : USINT := 90; (*Fast servo speed*)
		iMaxPosDev2UseLift : INT := 10;
		tiDropDelay : TIME := T#1ms;
		tiDropReadyDelay : TIME := T#500ms;
		iSafeElevatorPosStart : INT := 92; (*Positie waar de elevator pas mag zakken naar de drop positie*)
		iSafeElevatorPosStartVak : INT := 246;
		iSafeElevatorPosEndVak : INT := 443;
		iSafeElevatorPosEnd : INT := 530;
		tiBunchBeltPulse : TIME := T#500ms;
		usTimingBU16 : USINT := 5; (*Pos=7*)
		usBunchBeltPosition : USINT;
	END_STRUCT;
	InterfaceBU : 	STRUCT
		usNextChainInput : SINT; (*ID of the chain containing the next flower 255  for none*)
		bReset : BOOL;
		bEnable : BOOL;
		iReleasePos : INT := 125;
		iReceivePos : INT := 265;
		usServoSpeed : USINT := 10; (*Bos Unit default speed 0-100 %*)
		bHomeCmd : BOOL; (*Move to home*)
		Command : BU_Command_Enum := BU_CMD_Ready;
		Status : BU_Status_enum := BU_ST_DISABLED;
		usError : USINT;
		bEmptyCmd : BOOL;
		bEmptyPerm : BOOL;
		bManualUpCmd : BOOL;
		bManualCmd : BOOL;
		bManualDownCmd : BOOL;
		iManualPosition : INT := 500;
		usManualSpeed : USINT := 50;
		usStemTarget : USINT := 4;
		usStemCount : USINT;
		iSpeedBunchbelt : INT := 2700; (*90Hz*)
		tiDelayActivateBunchBelts : TIME := T#2150ms; (*150*)
		tiDelayActiveGripper : TIME := T#500ms; (*150*)
		bReadyForDrop : BOOL := FALSE;
		bSimulation : BOOL := FALSE;
		bToggleBunchBelt : BOOL := FALSE; (*Draai even de Bunch belt*)
		bManualGripperCmd : BOOL := FALSE; (*Aktiveer alle grippers*)
		bAddFlowerNow : BOOL := FALSE; (*Voeg voor test een bloem toe*)
		bFault : BOOL := TRUE; (*Hoog als er een fout is*)
	END_STRUCT;
	BunchUnit : 	STRUCT  (*Verzameling parameters bosunit*)
		typOUT : _buOUT;
		typIN : _buIN;
		usUnitNmbr : USINT := 0;
		usChainPos : USINT := 0;
		usErrorState : USINT := 99;
		typServo : Servo_typ;
		typInterface : InterfaceBU;
		typSettings : SettingsBU;
		typBunchBelts : AcpInverter_typ;
		motBunchBelts : ACPinverter;
		BunchBeltControl : TOF;
		GripperControl : TOF;
		rsActivateGripper : RS;
		bAddFlower : BOOL := FALSE;
		bBusyDrop : BOOL := FALSE;
	END_STRUCT;
	_buOUT : 	STRUCT
		bOnline : BOOL;
		bElevator : BOOL := FALSE;
		bActivateGripper : BOOL := FALSE;
		bBunchGripper : BOOL := FALSE;
		bReleaseGripper : BOOL := FALSE; (*Release load from gripper to conveyor*)
		GripperState : BU_Visu_Gripper_enum;
		ReleaseState : BU_Visu_Release_enum;
		ElevatorState : BU_Elevator_enum;
		bStopServo : BOOL := FALSE; (*Extra Stop uit I?O-Lijst*)
		bEndStageServo : BOOL := FALSE; (*idem*)
		bEnableServo : BOOL := FALSE; (*idem*)
	END_STRUCT;
	_buIN : 	STRUCT
		bOnline : BOOL;
		bPosHome : BOOL := FALSE;
		bElevatorUp : BOOL := FALSE;
		bElevatorMid : BOOL := FALSE;
		bElevatorDown : BOOL := FALSE;
		bTestUnit : BOOL := FALSE;
		bNegMove : BOOL := FALSE;
		bPosMove : BOOL := FALSE;
		ElevatorState : BU_Visu_Elevator_enum;
		in : ARRAY[0..7]OF BOOL; (*//Used for IO Handling (Fast task)*)
	END_STRUCT;
END_TYPE
```

#### BU.st - Operate Elevator
```iecst
(********************************************************************
 * COPYRIGHT --
 ********************************************************************
 * Program: BU
 * File: Lift.st
 * Author: ronspa
 * Created: September 25, 2014
 ********************************************************************
 * Implementation of program BU
 ********************************************************************)

(*Operate Elevator*)
FUNCTION Elevator
	IF (ThisBU.typServo.status.VAL2.diPosition >= ThisBU.typSettings.iSafeElevatorPosStart) AND
		(ThisBU.typServo.status.VAL2.diPosition <= ThisBU.typSettings.iSafeElevatorPosEnd) AND
		(ThisBU.typServo.status.VAL2.diPosition <= ThisBU.typSettings.iSafeElevatorPosStartVak OR
		ThisBU.typServo.status.VAL2.diPosition >= ThisBU.typSettings.iSafeElevatorPosEndVak) THEN
		ThisBU.typOUT.bElevator := DINT_TO_BOOL(bElevator);
		Elevator := TRUE;
	ELSE
		// Move Servo to save position
		// There should be a LOG here, this can not happen!!!!!!!!
		IF ThisBU.typInterface.iReleasePos < ThisBU.typSettings.iSafeElevatorPosStart THEN
			ThisBU.typInterface.iReleasePos := ThisBU.typSettings.iSafeElevatorPosStart + 10;
		ELSE
			IF ThisBU.typInterface.iReleasePos > ThisBU.typSettings.iSafeElevatorPosEnd THEN
				ThisBU.typInterface.iReleasePos := ThisBU.typSettings.iSafeElevatorPosEnd - 10;
			ELSE
				IF (ThisBU.typInterface.iReleasePos < ThisBU.typSettings.iSafeElevatorPosEndVak) AND (ThisBU.typInterface.iReleasePos > ThisBU.typSettings.iSafeElevatorPosStartVak) THEN
					IF ThisBU.typInterface.iReleasePos > (ThisBU.typSettings.iSafeElevatorPosStartVak + (ThisBU.typSettings.iSafeElevatorPosEndVak - ThisBU.typSettings.iSafeElevatorPosStartVak) /2) THEN
						ThisBU.typInterface.iReleasePos := ThisBU.typSettings.iSafeElevatorPosEndVak + 10;
					ELSE
						ThisBU.typInterface.iReleasePos := ThisBU.typSettings.iSafeElevatorPosStartVak - 10;
					END_IF
				END_IF
			END_IF
		END_IF
		ServoMovePosition(ThisBU, ThisBU.typInterface.iReleasePos, 45);
	END_IF
END_FUNCTION

FUNCTION CheckTimers
	tonElevator(IN := (ThisBU.typOUT.bElevator AND NOT ThisBU.typIN.bElevatorUp) OR (ThisBU.typOUT.bElevator AND NOT ThisBU.typIN.bElevatorDown), PT := T#1s);

	IF (tonElevator.Q) THEN
		// Time out
		CheckTimers := BU_ST_TIMEOUT_LIFT;
		RETURN;
	END_IF
	CheckTimers := Status;
END_FUNCTION

FUNCTION DefaultSettingsBU
	ThisBU.typSettings.usHomeSpeed 			:= iHS;
	ThisBU.typSettings.iMaxPosDev2UseLift 	:= iMPD2UL;
	ThisBU.typSettings.iReceivePos 			:= iRP;
	ThisBU.typSettings.iReleasePos 			:= iRlP;
	ThisBU.typSettings.usSpeed 				:= iSPD;
	ThisBU.typSettings.usFastSpeed 			:= iFSPD;
	ThisBU.typSettings.tiDropDelay 			:= tiDD;
	ThisBU.typSettings.tiDropReadyDelay 	:= tiDRD;
	ThisBU.typSettings.uiNextChainDelay 	:= uiNCD;
	ThisBU.typSettings.iSafeElevatorPosStart	:= iSEPStart;
	ThisBU.typSettings.iSafeElevatorPosStartVak	:= iSEPStartVak;
	ThisBU.typSettings.iSafeElevatorPosEndVak	:= iSEPEndVak;
	ThisBU.typSettings.iSafeElevatorPosEnd	:= iSEPEnd;
	ThisBU.typSettings.tiBunchBeltPulse	:= tiBBP;
END_FUNCTION

//Function call in IOpolling program (2ms)
FUNCTION ElevatorCil
	bElevatorUp_SR(SET1 := bUp, RESET := bMid OR bDown);

	//ThisBU.typIN.bElevatorUp := bElevatorUp_SR.Q1;

	bElevatorMid_SR(SET1 := bMid, RESET := bUp OR bDown);

	ThisBU.typIN.bElevatorMid := bElevatorMid_SR.Q1;

	bElevatorDown_SR(SET1 := bDown, RESET := bUp OR bMid);

	ThisBU.typIN.bElevatorDown := bElevatorDown_SR.Q1;
END_FUNCTION
```

### Library Logical/libraries_hav/PulsGen (IEC) - Pulsegenerator (variable High/Low pulse)

#### PulsGen.fun - Exported functions and function blocks
```iecst
(********************************************************************
 * COPYRIGHT --
 ********************************************************************
 * Library: PulsGen
 * File: PulsGen.fun
 * Author: jorkes
 * Created: July 18, 2014
 ********************************************************************
 * Functions and function blocks of library PulsGen
 ********************************************************************)

FUNCTION_BLOCK fbTriggerBuf
	VAR_INPUT
		CamPos : INT;
		reset : BOOL;
		trigger : BOOL;
		tiPuls : TIME;
		tiDelay : TIME;
		tiExtraLight : TIME;
	END_VAR
	VAR_OUTPUT
		outLight : BOOL;
		outCam : BOOL;
	END_VAR
	VAR
		tpPulsLight : TP;
		tpPulsCam : TP;
		tiOffset : TIME := T#30ms;
		tiActual : TIME;
		tiTime : TIME;
		tiStart : ARRAY[0..1] OF TIME;
		idx_1 : USINT;
		idx : USINT;
		idx_0 : USINT;
		zzEdge00000 : BOOL;
		zzEdge00001 : BOOL;
	END_VAR
END_FUNCTION_BLOCK

FUNCTION_BLOCK PulsGenerator
	VAR_INPUT
		tInit : BOOL;
		enable : BOOL;
		sysTim : DINT;
		tiHigh : TIME;
		tiLow : TIME;
	END_VAR
	VAR_OUTPUT
		bOutput : BOOL := FALSE;
	END_VAR
	VAR
		counter : USINT;
		time : DINT;
		state : USINT := 0;
		zzEdge00000 : BOOL;
	END_VAR
END_FUNCTION_BLOCK
```

#### PulsGen.st
```iecst
(********************************************************************
 * COPYRIGHT --
 ********************************************************************
 * Package: PulsGen
 * File: PulsGen.st
 * Author: jorkes
 * Created: July 18, 2014
 *******************************************************************)
FUNCTION_BLOCK PulsGenerator
	(* First time take over the systemtime *)
	IF EDGEPOS(tInit) THEN
		time := sysTim;
		state := 0;
		counter := 0;
	END_IF

	(* Run if enabled *)
	IF enable THEN
		CASE state OF
			(**)
			0:
				bOutput := TRUE;

				IF (sysTim - time) >= (TIME_TO_DINT(tiHigh)*1000) THEN
					state := 1;
					bOutput := FALSE;
					time := sysTim;
					counter := counter + 1;
				END_IF
			(**)
			1:
				bOutput := FALSE;

				IF ((sysTim - time) >= (TIME_TO_DINT(tiLow)*1000)) AND (counter < 16) THEN
					state := 0;
					bOutput := TRUE;
					time := sysTim;
				END_IF
		END_CASE;
	ELSE
		time := sysTim;
		state := 0;
	END_IF
END_FUNCTION_BLOCK

FUNCTION_BLOCK fbTriggerBuf
	IF EDGEPOS(reset) THEN
		idx := 0;
	END_IF

	IF EDGENEG(trigger) THEN
		IF idx = (CamPos-1) THEN
			tiTime := clock_ms();
		END_IF
		idx := (idx + 1) MOD 16;
	END_IF

	IF (clock_ms() - tiTime) >= tiDelay THEN
		tpPulsLight.IN := TRUE;
	ELSE
		tpPulsLight.IN := FALSE;
	END_IF

	IF (clock_ms() - tiTime) >= (tiDelay + tiExtraLight) THEN
		tpPulsCam.IN := TRUE;
	ELSE
		tpPulsCam.IN := FALSE;
	END_IF

	tpPulsLight(PT := tiPuls + tiExtraLight + tiExtraLight);
	tpPulsCam(PT := tiPuls);

	outLight := tpPulsLight.Q;
	outCam := tpPulsCam.Q;
END_FUNCTION_BLOCK
```

### Library Logical/libraries_hav/Servo (IEC) - Servo Drive (Festo Library)

#### Servo.fun - Exported functions and function blocks
```iecst
(********************************************************************
 * COPYRIGHT -- Microsoft
 ********************************************************************
 * Library: Servo
 * File: Servo.fun
 * Author: jorkes
 * Created: October 30, 2014
 ********************************************************************
 * Functions and function blocks of library Servo
 ********************************************************************)

FUNCTION ServoMovePosition : BOOL
	VAR_INPUT
		ThisBU : BunchUnit;
		NewPosition : INT;
		Speed : USINT;
	END_VAR
END_FUNCTION

FUNCTION ServoReset : BOOL
	VAR_INPUT
		ThisBU : BunchUnit;
	END_VAR
END_FUNCTION

FUNCTION ServoHome : BOOL
	VAR_INPUT
		ThisBU : BunchUnit;
	END_VAR
END_FUNCTION
```

#### Servo.typ - Exported data types
```iecst
(********************************************************************
 * COPYRIGHT --
 ********************************************************************
 * Library: BULib
 * File: Servo.typ
 * Author: ronspa
 * Created: September 29, 2014
 ********************************************************************
 * Data types of library BULib
 ********************************************************************)

TYPE
	stat_type : 	STRUCT
		SCON : SCON_status_typ;
		SPOS : SPOS_status_typ;
		SDIR : SDIR_status_typ;
		VAL2 : VAL2_stat_type;
		VAL1 : VAL1_stat_type;
	END_STRUCT;
	SPOS_status_typ : 	STRUCT
		bHALT : BOOL; (*Halt*)
		bACK : BOOL; (*Acknowledge start*)
		bMC : BOOL; (*Motion complete*)
		bTEACH : BOOL; (*Acknowledge Teach/Sampling*)
		bMOV : BOOL; (*Axis is moving*)
		bDEV : BOOL; (*Drag (deviation) error*)
		bSTILL : BOOL; (*Standstill control*)
		bREF : BOOL; (*Axis is referenced*)
		uiSPOS : USINT; (*Status byte*)
	END_STRUCT;
	PARA2_command_typ : 	STRUCT
		diPosition : DINT; (*Velocity as percentage of base value*)
	END_STRUCT;
	VAL1_stat_type : 	STRUCT
		usVelocity : USINT;
	END_STRUCT;
	SDIR_status_typ : 	STRUCT
		bABS : BOOL; (*Absolute/relative*)
		bCOM1 : BOOL; (*Control mode feedback*)
		bCOM2 : BOOL;
		bFNUM1 : BOOL; (*Function number feedback*)
		bFNUM2 : BOOL;
		bFGRP1 : BOOL; (*Function group feedback*)
		bFGRP2 : BOOL;
		bFUNC : BOOL; (*Function feedback*)
		uiSDIR : USINT; (*Status byte*)
	END_STRUCT;
	SCON_status_typ : 	STRUCT
		bENABLED : BOOL; (*Drive enabled*)
		bOPEN : BOOL; (*Operation enabled*)
		bWARN : BOOL; (*Warning*)
		bFAULT : BOOL; (*Fault*)
		b24VL : BOOL; (*Supply voltage is applied*)
		bLOCK : BOOL; (*Drive control by software*)
		bOPM1 : BOOL; (*Display operating mode*)
		bOPM2 : BOOL; (*Display operating mode*)
		uiSCON : USINT; (*Status byte*)
	END_STRUCT;
	Servo_typ : 	STRUCT
		enumServoState : SERVO_Status_enum := SERVO_READY;
		command : com_typ;
		status : stat_type;
		packed : Servo_packed_typ;
		enumServoCmd : SERVO_CMD_Enum := SERVO_CMD_READY;
		bOnLine : BOOL; (*Servo online*)
		usNode : USINT;
		SDO : SDO_type;
	END_STRUCT;
	CDIR_command_typ : 	STRUCT
		bABS : BOOL; (*Absolute/relative*)
		bCOM1 : BOOL; (*Control mode feedback*)
		bCOM2 : BOOL;
		bFNUM1 : BOOL; (*Function number feedback*)
		bFNUM2 : BOOL;
		bFGRP1 : BOOL; (*Function group feedback*)
		bFGRP2 : BOOL;
		bFUNC : BOOL; (*Function feedback*)
	END_STRUCT;
	CPOS_command_typ : 	STRUCT
		bHALT : BOOL; (*Halt*)
		bSTART : BOOL; (*Start positioning task*)
		bHOM : BOOL; (*Start homing*)
		bJOGP : BOOL; (*Jog positive*)
		bJOGN : BOOL; (*Job negative*)
		bTEACH : BOOL; (*Teach actual value*)
		bCLEAR : BOOL; (*Clear remaing position*)
		bNU : BOOL; (*Not used*)
	END_STRUCT;
	com_typ : 	STRUCT
		CCON : CCON_command_typ;
		CPOS : CPOS_command_typ;
		CDIR : CDIR_command_typ;
		PARA1 : PARA1_command_typ;
		PARA2 : PARA2_command_typ;
	END_STRUCT;
	Servo_packed_typ : 	STRUCT
		CCON : USINT; (*Control byte 1*)
		CPOS : USINT; (*Control byte 2*)
		CDIR : USINT; (*Control byte 3*)
		PARA1 : USINT; (*Control byte 4*)
		PARA2 : DINT; (*Control bytes 5-8*)
		SCON : USINT; (*Status byte 1*)
		SPOS : USINT; (*Status byte 2*)
		SDIR : USINT; (*Status byte 3*)
		VAL2 : DINT;
		VAL1 : USINT;
	END_STRUCT;
	CCON_command_typ : 	STRUCT
		bENABLE : BOOL; (*Drive enabled*)
		bSTOP : BOOL; (*Stop*)
		bBRAKE : BOOL; (*Open brake*)
		bRESET : BOOL; (*Reset fault*)
		bNU : BOOL; (*Not used*)
		bLOCK : BOOL; (*Software access locked*)
		bOPM1 : BOOL; (*Select operating mode*)
		bOPM2 : BOOL;
	END_STRUCT;
	VAL2_stat_type : 	STRUCT
		diPosition : DINT;
	END_STRUCT;
	PARA1_command_typ : 	STRUCT
		usVelocity : USINT; (*Velocity as percentage of base value*)
	END_STRUCT;
	SERVO_Status_enum :
		(
		SERVO_READY := 1,
		SERVO_HOMING_COMPLETE := 2,
		SERVO_WARNING := 3,
		SERVO_FAULT := 4,
		SERVO_HOMING_NOT_COMPLETED := 5,
		SERVO_IS_HOMING := 6,
		SERVO_RUNNING := 7,
		SERVO_DISABLED := 8
		);
	SERVO_CMD_Enum :
		(
		SERVO_CMD_HOME := 10,
		SERVO_CMD_RUN := 20,
		SERVO_CMD_RESET := 99,
		SERVO_CMD_READY := 100
		);
END_TYPE
```

#### ServoHome.st
```iecst
(********************************************************************
 * COPYRIGHT --
 ********************************************************************
 * Package: Servo
 * File: ServoHome.st
 * Author: ronspa
 * Created: January 27, 2015
 *******************************************************************)

FUNCTION ServoHome
	IF ThisBU.typServo.bOnLine THEN
		ThisBU.typServo.enumServoCmd := SERVO_CMD_HOME;
		ThisBU.typServo.command.PARA1.usVelocity := 10;
		ServoHome := TRUE;
	ELSE
		ServoHome := FALSE;
	END_IF
END_FUNCTION
```

#### ServoReset.st
```iecst
(********************************************************************
 * COPYRIGHT --
 ********************************************************************
 * Package: Servo
 * File: ServoReset.st
 * Author: ronspa
 * Created: January 27, 2015
 *******************************************************************)

FUNCTION ServoReset
	(* Insert code here *)
	//ThisBU.
	IF ThisBU.typServo.bOnLine THEN
		ThisBU.typServo.enumServoCmd := SERVO_CMD_RESET;
		ServoReset := TRUE;
	ELSE
		ServoReset := FALSE;
	END_IF
END_FUNCTION
```

#### ServoMovePosition.st
```iecst
(********************************************************************
 * COPYRIGHT --
 ********************************************************************
 * Program: Festo_Ref
 * File: FestoFun.st
 * Author: ronspa
 * Created: September 29, 2014
 *******************************************************************)

FUNCTION ServoMovePosition
	IF ThisBU.typServo.bOnLine AND ThisBU.typServo.enumServoCmd = SERVO_CMD_READY THEN
		IF ThisBU.typServo.command.PARA2.diPosition <> NewPosition THEN
			ThisBU.typServo.status.SPOS.bMC := FALSE;
		END_IF
		ThisBU.typServo.command.PARA2.diPosition := NewPosition;
		ThisBU.typServo.command.PARA1.usVelocity := Speed;
		ThisBU.typServo.enumServoCmd := SERVO_CMD_RUN;
		ServoMovePosition := TRUE;
		IF NOT ThisBU.typInterface.bManualCmd THEN
			ThisBU.typInterface.iManualPosition := NewPosition;
			ThisBU.typInterface.usManualSpeed := Speed;
		END_IF
	ELSE
		ServoMovePosition := FALSE;
	END_IF
END_FUNCTION
```

### Library Logical/libraries_hav/SDO (IEC) - CAN SDO Read/Write Library

#### SDO.st
```iecst
(********************************************************************
 * COPYRIGHT --
 ********************************************************************
 * Package: BULib
 * File: SDO.st
 * Author: jorkes
 * Created: October 07, 2014
 *******************************************************************)
FUNCTION SDO_Servo
			// Als Command = 1 (=READ_SDO) dan spring naar step 40 en voert functie readSDO uit
	CASE Command OF
		SERVO_WR : // 1
			Step := 10;
			Command := 99;
		SERVO_RD : // 2
			Step := 20;
			Command := 99;
		STANDBY : // Standby
	END_CASE

	CASE Step OF
		//-----------------------------------------------------------
		// Servo write SDO
		//-----------------------------------------------------------
		10:
			ThisBU.typServo.SDO.Write.enable := TRUE;
			ThisBU.typServo.SDO.Write.pDevice := ADR('SS1.IF1');
			ThisBU.typServo.SDO.Write.node := Node;
			ThisBU.typServo.SDO.Write.index := Index;
			ThisBU.typServo.SDO.Write.subIndex := SubIndex;
			ThisBU.typServo.SDO.Write.dataCount := 4;

			// Wait for function is done, OK or error
			IF (ThisBU.typServo.SDO.Write.status = ERR_OK) THEN
				ThisBU.typServo.SDO.Write.pData := ADR(ThisBU.typServo.SDO.udDataWrite[0]);
				Step := 0;
			ELSIF (ThisBU.typServo.SDO.Write.status <> ERR_FUB_BUSY) THEN
				Error := ThisBU.typServo.SDO.Write.status;
				Step := 100; 	// STATE_ERROR;
			END_IF

			ThisBU.typServo.SDO.Write();
		//-----------------------------------------------------------
		// Servo read SDO
		//-----------------------------------------------------------
		20:
			ThisBU.typServo.SDO.Read.enable := TRUE;
			ThisBU.typServo.SDO.Read.pDevice := ADR('SS1.IF1');
			ThisBU.typServo.SDO.Read.node := Node;
			ThisBU.typServo.SDO.Read.index := Index;
			ThisBU.typServo.SDO.Read.subIndex := SubIndex;
			ThisBU.typServo.SDO.Read.dataCount := 4;
			ThisBU.typServo.SDO.Read.pData := ADR(ThisBU.typServo.SDO.udDataRead[0]);
			ThisBU.typServo.SDO.Read();

			// Wait for function is done, OK or error
			IF (ThisBU.typServo.SDO.Read.status = ERR_OK) THEN
				Step := 0;
			ELSIF (ThisBU.typServo.SDO.Read.status <> ERR_FUB_BUSY) THEN
				Error := ThisBU.typServo.SDO.Read.status;
				Step := 100; 	// STATE_ERROR;
			END_IF

			SDO_Servo := ThisBU.typServo.SDO.udDataRead[0];
		// Error
		//-----------------------------------------------------------
		100:
	END_CASE
END_FUNCTION

FUNCTION SDO_Inverter
			// Als Command = 1 (=READ_SDO) dan spring naar step 40 en voert functie readSDO uit
	CASE Command OF
		INV_WR	 : // 3
			Step := 30;
			Command := 99;
		INV_RD	 : // 4
			Step := 40;
			Command := 99;
		STANDBY : // Standby
	END_CASE

	(*CASE Step OF
		//-----------------------------------------------------------
		// Inverter write SDO
		//-----------------------------------------------------------
		30:
			typBunchBelts[i].SDO.Write.enable := TRUE;
			typBunchBelts[i].SDO.Write.pDevice := ADR('SS1.IF1');
			typBunchBelts[i].SDO.Write.node := Node;
			typBunchBelts[i].SDO.Write.index := Index;
			typBunchBelts[i].SDO.Write.subIndex := SubIndex;
			typBunchBelts[i].SDO.Write.dataCount := 2;

			// Wait for function is done, OK or error
			//IF (ThisBU.typServo.SDO.Write.status = ERR_OK) THEN
			IF (typBunchBelts[i].SDO.Write.status = ERR_OK) THEN
				typBunchBelts[i].SDO.Write.pData := ADR(typBunchBelts[i].SDO.udDataWrite[0]);
				Step := 0;
			ELSIF (ThisMotor.typBunchBelts.SDO.Write.status <> ERR_FUB_BUSY) THEN
				Error := typBunchBelts[i].SDO.Write.status;
				Step := 100; 	// STATE_ERROR;
			END_IF

			ThisMotor.typBunchBelts.SDO.Write();
		//-----------------------------------------------------------
		// Inverter read SDO
		//-----------------------------------------------------------
		40:
			typBunchBelts[i].SDO.Read.enable := TRUE;
			typBunchBelts[i].SDO.Read.pDevice := ADR('SS1.IF1');
			typBunchBelts[i].SDO.Read.node := Node;
			typBunchBelts[i].SDO.Read.index := Index;
			typBunchBelts[i].SDO.Read.subIndex := SubIndex;
			typBunchBelts[i].SDO.Read.dataCount := 2;
			typBunchBelts[i].SDO.Read.pData := ADR(ThisMotor.typBunchBelts.SDO.udDataRead[0]);
			typBunchBelts[i].SDO.Read();

			// Wait for function is done, OK or error
			IF (typBunchBelts[i].SDO.Read.status = ERR_OK) THEN
				Step := 0;
			ELSIF (typBunchBelts[i].SDO.Read.status <> ERR_FUB_BUSY) THEN
				Error := ThisMotor.typBunchBelts.SDO.Read.status;
				Step := 100; 	// STATE_ERROR;
			END_IF

			SDO_Inverter := typBunchBelts[i].SDO.udDataRead[0];
		// Error
		//-----------------------------------------------------------
		100:

	END_CASE*)
END_FUNCTION
```

#### SDO.fun - Exported functions and function blocks
```iecst
(********************************************************************
 * COPYRIGHT -- Microsoft
 ********************************************************************
 * Library: SDO
 * File: SDO.fun
 * Author: jorkes
 * Created: October 30, 2014
 ********************************************************************
 * Functions and function blocks of library SDO
 ********************************************************************)

FUNCTION SDO_Servo : UDINT
	VAR_INPUT
		ThisBU : BunchUnit;
		Node : USINT;
		Index : UDINT;
		SubIndex : UDINT;
		Command : NodeState_enum := STANDBY;
	END_VAR
	VAR
		Error : UINT;
		Step : USINT;
	END_VAR
END_FUNCTION

FUNCTION SDO_Inverter : UDINT
	VAR_INPUT
		i : USINT;
		Node : USINT;
		Index : UDINT;
		SubIndex : UDINT;
		Command : NodeState_enum := STANDBY;
	END_VAR
	VAR
		Error : UINT;
		Step : USINT;
	END_VAR
END_FUNCTION
```

#### SDO.typ - Exported data types
```iecst
(********************************************************************
 * COPYRIGHT --
 ********************************************************************
 * Library: BULib
 * File: SDO.typ
 * Author: jorkes
 * Created: October 07, 2014
 ********************************************************************
 * Data types of library BULib
 ********************************************************************)

TYPE
	NodeState_enum :
		(
		SERVO_WR := 1,
		SERVO_RD := 2,
		INV_WR := 3,
		INV_RD := 4,
		STANDBY := 99
		);
	SDO_type : 	STRUCT
		udIndex : UDINT;
		udSubIndex : UDINT;
		usNode : USINT;
		Write : nxcomSdoWrite;
		udDataWrite : ARRAY[0..3]OF UDINT;
		Read : nxcomSdoRead;
		udDataRead : ARRAY[0..3]OF UDINT;
	END_STRUCT;
END_TYPE
```

### Library Logical/libraries_hav/Lichtkrant (IEC) - Lichtkrant functies
Depends on: standard

#### Lichtkrant.st
```iecst
(********************************************************************
 * COPYRIGHT -- Microsoft
 ********************************************************************
 * Package: Lichtkrant
 * File: Lichtkrant.st
 * Author: jorkes
 * Created: November 20, 2014
 *******************************************************************)
FUNCTION_BLOCK fbSetText
	(* Lichtkrant *)
	(**********************************************************************
		Identification:
			FUNCTION block	:	setText
			Description		:	Convert text to Lichtkrant text with checksum

	(*----------------------------------------------------------------------
	 	Declaration;
			ThisData	= INPUT[DataPackage] = Select lichtkrant
			text 		= INPUT[STRING[80]]	 = String input

	(**********************************************************************)
	ThisData.methodSpeed := interval;
	ThisData.laggingCom := presentation;
	ThisData.fontCode := font;
	ThisData.colorCode := color;

	_param := CONCAT(ThisData.lineNumber, ThisData.pageNumber);
	_param := CONCAT(_param, ThisData.leadingCom);
	_param := CONCAT(_param, ThisData.methodSpeed);
	_param := CONCAT(_param, ThisData.waitingTime);
	_param := CONCAT(_param, ThisData.laggingCom);
	_param := CONCAT(_param, ThisData.fontCode);
	_param := CONCAT(_param, ThisData.colorCode);

	_param := CONCAT(_param, IN);

	_buflen := LEN(_param);

	// string omzetten naar USINT array
	brsmemcpy(ADR(_array), ADR(_param), SIZEOF(_array));

	_sum := 0;

	FOR _idx := 0 TO (_buflen - 1) DO
		_sum := _sum XOR _array[_idx];
	END_FOR

	dec2hex_0(usMaxHexDigit := 2, udInputDec := _sum);

	_hexSum := dec2hex_0.strOutputHex;

	IF (LEFT(_hexSum, 1) = '0') THEN //LEFT(string, count)
		IF (LEFT(_hexSum, 2) = '00') THEN
			_hexSum := DELETE(_hexSum, 2, 1); //DELETE(string, index, position)
		ELSE
			_hexSum := DELETE(_hexSum,1, 1);
		END_IF
	END_IF

	_param := CONCAT('<ID00>', _param);
	_param := CONCAT(_param, _hexSum);
	_param := CONCAT(_param, '<E>');

	OUT := _param;
END_FUNCTION_BLOCK
```

#### Lichtkrant.typ - Exported data types
```iecst
(********************************************************************
 * COPYRIGHT -- Microsoft
 ********************************************************************
 * Library: Lichtkrant
 * File: Lichtkrant.typ
 * Author: jorkes
 * Created: November 17, 2014
 ********************************************************************
 * Data types of library Lichtkrant
 ********************************************************************)

TYPE
	_methodSpeed : 	STRUCT
		fast : STRING[4] := '<MA>';
		middle : STRING[4] := '<MQ>';
		slow : STRING[4] := '<Ma>';
	END_STRUCT;
	_laggingCom : 	STRUCT
		normal : STRING[4] := '<FK>';
		upDown : STRING[4] := '<FJ>';
		horizontalScroll : STRING[4] := '<FF>';
	END_STRUCT;
	DataPackage : 	STRUCT
		lineNumber : STRING[4] := '<L1>';
		pageNumber : STRING[4] := '<PA>';
		leadingCom : STRING[4] := '<FA>';
		methodSpeed : STRING[4] := '<MA>';
		waitingTime : STRING[4] := '<WA>';
		methodSpeed_ : _methodSpeed := (fast:='<MA>',middle:='<MQ>',slow:='<Ma>');
		laggingCom_ : _laggingCom := (normal:='<FK>',upDown:='<FJ>',horizontalScroll:='<FF>');
		laggingCom : STRING[4] := '<FK>';
		fontCode : STRING[4] := '<CC>';
		colorCode : STRING[4] := '<AA>';
		fontCode_ : _fontCode := (narowSize_4x7:='<AC>',boldSize_6x7:='<AB>',normalSize_5x7:='<AA>');
		colorCode_ : _colorCode := (Yellow:='<CJ>',brightOrange:='<CI>',brightGreen:='<CF>',brightRed:='<CC>');
	END_STRUCT;
	_fontCode : 	STRUCT
		narowSize_4x7 : STRING[4] := '<AC>';
		boldSize_6x7 : STRING[4] := '<AB>';
		normalSize_5x7 : STRING[4] := '<AA>';
	END_STRUCT;
	_colorCode : 	STRUCT
		Yellow : STRING[4] := '<CJ>';
		brightOrange : STRING[4] := '<CI>';
		brightGreen : STRING[4] := '<CF>';
		brightRed : STRING[4] := '<CC>';
	END_STRUCT;
END_TYPE
```

#### Lichtkrant.fun - Exported functions and function blocks
```iecst
(********************************************************************
 * COPYRIGHT -- Microsoft
 ********************************************************************
 * Library: Lichtkrant
 * File: Lichtkrant.fun
 * Author: jorkes
 * Created: November 17, 2014
 ********************************************************************
 * Functions and function blocks of library Lichtkrant
 ********************************************************************)

FUNCTION_BLOCK fbSetText
	VAR_INPUT
		ThisData : DataPackage;
		IN : STRING[80]; (*//Data string*)
		color : STRING[4] := '<CC>';
		font : STRING[4] := '<AC>';
		interval : STRING[4] := '<MA>';
		presentation : STRING[4] := '<FK>';
	END_VAR
	VAR_OUTPUT
		OUT : STRING[100];
	END_VAR
	VAR
		dec2hex_0 : dec2hex;
		_param : STRING[80];
		_idx : UINT;
		_array : ARRAY[0..255] OF USINT;
		_hexSum : STRING[4];
		_sum : UINT;
		_buflen : UINT;
	END_VAR
END_FUNCTION_BLOCK
```

### Library Logical/libraries_hav/Chain (IEC) - Chain Indicator

#### Chain.typ - Exported data types
```iecst
(********************************************************************
 * COPYRIGHT -- Microsoft
 ********************************************************************
 * Library: Chain
 * File: Chain.typ
 * Author: jorkes
 * Created: November 18, 2014
 ********************************************************************
 * Data types of library Chain
 ********************************************************************)

TYPE
	_cntrs : 	STRUCT
		usChainCounter : USINT; (*0-75*)
		uiChainCnt16x16 : UINT; (*0-255*)
		usChainOffset : USINT; (*0-75*)
		bStartChainCntr : BOOL;
		usStartUpCntr : USINT;
	END_STRUCT;
	Shiftregister : {REDUND_UNREPLICABLE} 	STRUCT  (*Schuifregister*)
		typEncoder : {REDUND_UNREPLICABLE} _encoder;
		typGripper : {REDUND_UNREPLICABLE} ARRAY[0..74]OF _gripper;
		uiGripperCnt : {REDUND_UNREPLICABLE} USINT := 75; (*Aantal grijpers die fysiek in de machine zitten*)
		uiCameraPosition : {REDUND_UNREPLICABLE} ARRAY[0..3]OF USINT := [2,3,4,5]; (*Positie in schuifregister waar Camera's hangen*)
		uiRejectPosition : {REDUND_UNREPLICABLE} USINT := 9;
		uiBunchUnitPosition : {REDUND_UNREPLICABLE} ARRAY[0..20]OF USINT := [11,14,16,18,20,23,25,27,30,32,0,0,0,0,0,0,0,0,0,0,0]; (*Positie bosstations t.o.v. de ketting (grijpers)*)
		tiDistanceBetweenGrippers : {REDUND_UNREPLICABLE} TIME := T#600ms; (*Tijd tussen twee grijpers*)
		reGripperSpeed_CmSec : {REDUND_UNREPLICABLE} REAL := 0.0; (*Snelheid van de grijpers in cm/sec*)
		reChainlength : {REDUND_UNREPLICABLE} REAL; (*Ketting lengte*)
		reGripperDistanceBetween_mm : {REDUND_UNREPLICABLE} REAL := 304.88; (*Aantal mm tussen de grijpers*)
		uiMachineSpeed : {REDUND_UNREPLICABLE} UINT := 6000; (*Machine snelheid in grijpers per uur*)
		typCounters : {REDUND_UNREPLICABLE} _cntrs;
	END_STRUCT;
	_encoder : {REDUND_UNREPLICABLE} 	STRUCT
		uiEncSensorPosition1 : {REDUND_UNREPLICABLE} UINT := 0; (*Schuifregisterpositie1*)
		uiEncSensorPosition2 : {REDUND_UNREPLICABLE} UINT := 34; (*Schuifregisterpositie2*)
		tiEncBetween : {REDUND_UNREPLICABLE} TIME := T#0S; (*Tijd tussen de twee encoder sensoren*)
		reGrippersBetween : {REDUND_UNREPLICABLE} REAL := 0.0; (*Aantal grijpers tussen de twee encoder sensoren*)
		reDistanceBetween : {REDUND_UNREPLICABLE} REAL := 0.0; (*Afstand tussen de twee encoder sensoren*)
	END_STRUCT;
	_gripper : {REDUND_UNREPLICABLE} 	STRUCT
		usSetTarget : {REDUND_UNREPLICABLE} SINT := -2; (*-2=Empty, -1=Reject 0..x BosUnit*)
		uiCorrection : {REDUND_UNREPLICABLE} UINT := 0;
		uiLength : {REDUND_UNREPLICABLE} UINT := 0;
		uiWeight : {REDUND_UNREPLICABLE} UINT := 0;
		uiTimingBU16 : {REDUND_UNREPLICABLE} UINT := 0; (*Timing from command*)
		bRejectActive : {REDUND_UNREPLICABLE} BOOL := FALSE; (*TRUE if bRejectOnOff is valid*)
		bRejectOnOff : {REDUND_UNREPLICABLE} BOOL := FALSE; (*if Target = -1, set/reset reject*)
		siEmptyBU : {REDUND_UNREPLICABLE} SINT := -2; (*Emprty BU *)
		bFast : {REDUND_UNREPLICABLE} BOOL := FALSE; (*Fast servo movement*)
	END_STRUCT;
END_TYPE
```

#### Chain.fun - Exported functions and function blocks
```iecst
(********************************************************************
 * COPYRIGHT -- Microsoft
 ********************************************************************
 * Library: Chain
 * File: Chain.fun
 * Author: jorkes
 * Created: November 18, 2014
 ********************************************************************
 * Functions and function blocks of library Chain
 ********************************************************************)

FUNCTION_BLOCK fbAverage
	VAR_INPUT
		enable : BOOL;
		index : USINT;
		tiMeasure : TIME;
	END_VAR
	VAR_OUTPUT
		tiAverage : TIME;
	END_VAR
	VAR
		_tiMusecDiff1 : ARRAY[0..9] OF TIME;
		idx : USINT := 0;
		size : USINT := 0;
	END_VAR
END_FUNCTION_BLOCK

FUNCTION fbChainlength : REAL
	VAR_INPUT
		ThisSHIFTREG : Shiftregister;
	END_VAR
END_FUNCTION

FUNCTION fbGripperSpeed : REAL
	VAR_INPUT
		ThisSHIFTREG : Shiftregister;
	END_VAR
END_FUNCTION

FUNCTION fbEncoderDistance : REAL
	VAR_INPUT
		ThisSHIFTREG : Shiftregister;
	END_VAR
END_FUNCTION

FUNCTION fbGripperDistance : REAL
	VAR_INPUT
		ThisSHIFTREG : Shiftregister;
	END_VAR
END_FUNCTION

FUNCTION fbEncoderBetween : TIME
	VAR_INPUT
		ThisSHIFTREG : Shiftregister;
		tiBetween : TIME;
	END_VAR
END_FUNCTION

FUNCTION fbResetGripper : BOOL
	VAR_INPUT
		ThisGripper : _gripper;
	END_VAR
END_FUNCTION
```

#### Chain.st
```iecst
(********************************************************************
 * COPYRIGHT -- Microsoft
 ********************************************************************
 * Package: Chain
 * File: Chain.st
 * Author: jorkes
 * Created: November 18, 2014
 *******************************************************************)
FUNCTION_BLOCK fbAverage
	tiAverage := 0;

	size := ( SIZEOF(_tiMusecDiff1)/SIZEOF(_tiMusecDiff1[0]) );
	index := index MOD size;

	_tiMusecDiff1[index] := tiMeasure;

	IF enable THEN
		FOR idx := 0 TO (size-1) DO
			//Assign timestamp of sensor puls length
			tiAverage := tiAverage + _tiMusecDiff1[idx];
		END_FOR

		//Everage of 10 sensor pulses
		tiAverage := tiAverage / size;
	END_IF
END_FUNCTION_BLOCK

FUNCTION fbChainlength
	ThisSHIFTREG.reChainlength := (UINT_TO_REAL(ThisSHIFTREG.uiGripperCnt)*ThisSHIFTREG.reGripperDistanceBetween_mm)/1000;
	//fbChainlength := ThisSHIFTREG.reChainlength;
END_FUNCTION

FUNCTION fbGripperSpeed
	ThisSHIFTREG.reGripperSpeed_CmSec := (ThisSHIFTREG.reGripperDistanceBetween_mm/10)*UINT_TO_REAL(ThisSHIFTREG.uiMachineSpeed)/3600;
	//fbGripperSpeed := ThisSHIFTREG.reGripperSpeed_CmSec;
END_FUNCTION

FUNCTION fbEncoderDistance
	ThisSHIFTREG.typEncoder.reDistanceBetween := ( (TIME_TO_REAL(ThisSHIFTREG.typEncoder.tiEncBetween)/1000)*ThisSHIFTREG.reGripperSpeed_CmSec )/100;
	//fbEncoderDistance := ThisSHIFTREG.typEncoder.reDistanceBetween;
END_FUNCTION

FUNCTION fbGripperDistance
	ThisSHIFTREG.typEncoder.reGrippersBetween := ThisSHIFTREG.typEncoder.reDistanceBetween/(ThisSHIFTREG.reGripperDistanceBetween_mm/1000);
	//fbGripperDistance := ThisSHIFTREG.typEncoder.reGrippersBetween;
END_FUNCTION

FUNCTION fbEncoderBetween
	ThisSHIFTREG.typEncoder.tiEncBetween := tiBetween;
	//fbEncoderBetween := ThisSHIFTREG.typEncoder.tiEncBetween;
END_FUNCTION

FUNCTION fbResetGripper
	/////ThisGripper.siEmptyBU := -2;
	//ThisGripper.bRejectActive := FALSE;
	//ThisGripper.bRejectOnOff := FALSE;
	//ThisGripper.uiCorrection := 0;
	ThisGripper.uiLength := 0;
	ThisGripper.uiTimingBU16 := 0;
	ThisGripper.uiWeight := 0;
	ThisGripper.usSetTarget := -2;
END_FUNCTION
```

### Library Logical/libraries_hav/hex2dec (IEC, version 0.02.0)
Depends on: AsString, AsString, runtime, standard

#### hex2dec.fun
```iecst
FUNCTION_BLOCK hex2dec
	VAR_INPUT
		Hexadecimal : STRING[8];
	END_VAR
	VAR_OUTPUT
		Decimal : DINT;
	END_VAR
	VAR
		Dyn_Usint : REFERENCE TO USINT;
		dMemcmpResult : DINT;
		strHexOld : STRING[8];
		strHexChar : STRING[2];
		i : INT;
		iStringLenght : INT;
	END_VAR
END_FUNCTION_BLOCK

FUNCTION_BLOCK dec2hex
	VAR_INPUT
		usMaxHexDigit : USINT;
		udInputDec : UDINT;
	END_VAR
	VAR_OUTPUT
		strOutputHex : STRING[8];
	END_VAR
	VAR
		udMask : UDINT;
		usIndex : USINT;
		udDec : ARRAY[0..7] OF UDINT;
		udDecimal : UDINT;
		lenHex : USINT;
		strHex : ARRAY[0..7] OF STRING[1];
		udOldInputDec : UDINT;
		udResult : UDINT;
	END_VAR
END_FUNCTION_BLOCK
```

#### dec2hex.st
```iecst
FUNCTION_BLOCK dec2hex
	(* Implementation of dec2hex *)
	(**********************************************************************
		Identification:
			Function block:	dec2hex
			Description		:	Convertor from decimal to hexidecimal
	(*----------------------------------------------------------------------
		History:
			Version			date				author	description
			0.01				28-9-2005		HD			First release
			0.02				26-7-2010		HD			More Hex numbers max 7 (UDINT input)

	(*----------------------------------------------------------------------
	 	Declaration;
			usMaxHexDigit	= INPUT[USINT] 		= Number of Hex digits
			udInputDec 		= INPUT[UINT]		= decimal input
			Hexadecimal 	= OUTPUT[STRING(2)] = hexadecimal output

	(**********************************************************************)

IF (udInputDec <> udOldInputDec) THEN
	udOldInputDec := udInputDec;

	IF (usMaxHexDigit > 7) THEN
 		usMaxHexDigit := 7;
	END_IF

	udMask := 16#0000000F;
	strOutputHex := '';
	FOR usIndex := 0 TO usMaxHexDigit	DO

		IF (usIndex = 0) THEN
			udDec[usIndex] := udInputDec AND udMask;
		ELSE
			udMask := SHL(udMask,4);
			udDec[usIndex] := SHR(udInputDec AND udMask,usIndex*4);
		END_IF

		udDecimal := (udDec[usIndex] MOD 16);

		CASE udDecimal OF
		 10: strHex[usMaxHexDigit-usIndex] := 'A';
		 11: strHex[usMaxHexDigit-usIndex] := 'B';
		 12: strHex[usMaxHexDigit-usIndex] := 'C';
		 13: strHex[usMaxHexDigit-usIndex] := 'D';
		 14: strHex[usMaxHexDigit-usIndex] := 'E';
		 15: strHex[usMaxHexDigit-usIndex] := 'F';
		ELSE
			itoa(udDecimal, ADR(strHex[usMaxHexDigit-usIndex]));
		END_CASE
		strcat(ADR(strOutputHex), ADR(strHex[usIndex]));

	END_FOR
END_IF

END_FUNCTION_BLOCK
```

#### hex2dec.st
```iecst
FUNCTION_BLOCK hex2dec
	(* Implementation of hex2dec *)
	(**********************************************************************
		Identification:
			Function block:	hex2dec
			Description		:	Convertor from hexidecimal to decimal
	(*----------------------------------------------------------------------
		History:
			Version			date					author	description
			0.01				03-04-2007		HD			First release

	(*----------------------------------------------------------------------
	 	Declaration;
			Hexadecimal = INPUT[STRING(8)] 	= hexadecimal input
			Decimal 		= INPUT[DINT]				= decimal output

	(**********************************************************************)

	dMemcmpResult := memcmp(ADR(Hexadecimal), ADR(strHexOld), SIZEOF(Hexadecimal));
	IF (dMemcmpResult <> 0) THEN
		Decimal := 0;
		iStringLenght := LEN(Hexadecimal);;
		i := iStringLenght - 1;
		IF (iStringLenght > 0) THEN

			WHILE i > -1 DO
				Dyn_Usint ACCESS(ADR(Hexadecimal) + i);

				(* Convert ASCI code to decimal *)
				CASE Dyn_Usint OF
					48:			strHexChar := '0';
					49:			strHexChar := '1';
					50:			strHexChar := '2';
					51:			strHexChar := '3';
					52:			strHexChar := '4';
					53:			strHexChar := '5';
					54:			strHexChar := '6';
					55:			strHexChar := '7';
					56:			strHexChar := '8';
					57:			strHexChar := '9';
					65,97:	strHexChar := '10';
					66,98:	strHexChar := '11';
					67,99:	strHexChar := '12';
					68,100:	strHexChar := '13';
					69,101:	strHexChar := '14';
					70,102:	strHexChar := '15';
				END_CASE

				(* Formule to calulate hex to decimal *)
				Decimal := Decimal + ( (atoi(ADR(strHexChar))) * REAL_TO_DINT( EXPT(16, (iStringLenght-1-i))) );

				i := i - 1;

			END_WHILE
		END_IF
	END_IF
	strHexOld := Hexadecimal;

END_FUNCTION_BLOCK
```

### Library Logical/libraries_hav/Serial (IEC) - Library for RS232 communication

#### Serial.typ - Exported data types
```iecst
(********************************************************************
 * COPYRIGHT -- Microsoft
 ********************************************************************
 * Library: Serial
 * File: Serial.typ
 * Author: jorkes
 * Created: November 26, 2014
 ********************************************************************
 * Data types of library Serial
 ********************************************************************)
(*Enumeration for Statemachine*)

TYPE
	enSEND_STEPS :
		(
		FRM_WAIT := 0, (*Defines the wait step*)
		FRM_OPEN, (*Defines Step for FRM_xopen() *)
		FRM_GBUF, (*Defines Step for FRM_rbuf()*)
		FRM_ROBUF, (*Defines Step for FRM_robuf()*)
		FRM_CLOSE, (*Defines Step for FRM_close()*)
		FRM_ERROR := 255 (*Defines Step for Errorhandling*)
		);
END_TYPE

(*Command data type*)

TYPE
	command_typ : 	STRUCT
		open_send : BOOL; (*Open serial port and send data*)
		close : BOOL; (*Close serial port*)
	END_STRUCT;
END_TYPE

(*Sender type*)

TYPE
	Sender_typ : 	STRUCT
		step : enSEND_STEPS := FRM_OPEN; (*Step of the Statemachine*)
		Commands : command_typ; (*Commandinterface*)
		send_data : STRING[80]; (*Send data*)
		FRM_xopen_0 : FRM_xopen; (*Functionblock FRM_xopen()*)
		xopenConfig : XOPENCONFIG; (*Configuration Type for FRM_xopen()*)
		FRM_gbuf_0 : FRM_gbuf; (*Functionblock FRM_gbuf()*)
		FRM_robuf_0 : FRM_robuf; (*Functionblock FRM_robuf()*)
		FRM_write_0 : FRM_write; (*Functionblock FRM_write)*)
		FRM_close_0 : FRM_close; (*Functionblock FRM_close()*)
	END_STRUCT;
END_TYPE
```

#### Serial.fun - Exported functions and function blocks
```iecst
(********************************************************************
 * COPYRIGHT -- Microsoft
 ********************************************************************
 * Library: Serial
 * File: Serial.fun
 * Author: jorkes
 * Created: November 26, 2014
 ********************************************************************
 * Functions and function blocks of library Serial
 ********************************************************************)

FUNCTION_BLOCK fbSerial
	VAR_INPUT
		enable : BOOL := TRUE;
		text : STRING[80];
	END_VAR
	VAR CONSTANT
		BUSY : UINT := 65535; (*Functionblock BUSY status*)
	END_VAR
	VAR
		Sender : Sender_typ := (0); (*Structure with all instances and variables*)
	END_VAR
END_FUNCTION_BLOCK
```
